# B&R Automation Studio project NAEUL004C00R13L518F00 (part 41)

#### Act_InputConfig.st
```iecst
(** 2019-04-09 **)
ACTION Act_InputConfig:

	(* Always Change If Project Change *)

	//Pass Data To Link
	tylocalPneu.In.bLinkDIConvClrSen := g_tyDInput.bConvClrSen;
	tylocalPneu.In.bConvPusherReachedRetSlw := g_tyPshrConv.bPshrRetAllwTrav;
	tylocalPneu.In.bLinkDIPusherRetRS := g_tyDInput.bPusherRetRS;
	tylocalPneu.In.eLinkLifterBtmStat := g_tyLifterBtm.eStat;
	tylocalPneu.In.eLinkLifterBtmStatus := g_tyLifterBtm.eStatus;
	tylocalPneu.In.eLinkLifter2Stat := g_tyLifter2.eStat;
	tylocalPneu.In.eLinkLifter2Status := g_tyLifter2.eStatus;

	//Pass Data To Internal Use
	tylocalPneu.In.bSafetyRelaySig 	 	 := g_tyDInput.bSafetyRlySig;
	tylocalPneu.In.udiRstErr := g_tyRstErr.udiReset;
	tylocalPneu.In.bPrep := g_tyNtParamCurr.bProjOutletShutPrep;
	tylocalPneu.In.bUISimu := g_tyUIOut.bSimuMod;
	tylocalPneu.In.bManual := g_tyUIOut.bMnlMod;
	tylocalPneu.In.bTwoCtrlIn := g_tyNtParamCurr.bOutShutterTwoCtrlIn;
	tylocalPneu.In.sProgNm := g_tyNtParamCurr.sOutShutterProgNm;
	tylocalPneu.In.bExtSen := g_tyDInput.bOutShutterCloseRS;
	tylocalPneu.In.bRetSen := g_tyDInput.bOutShutterOpenRS;
	tylocalPneu.In.tExtTO := g_tyNtParamCurr.tOutShutterExtTO;
	tylocalPneu.In.tRetTO := g_tyNtParamCurr.tOutShutterRetTO;
	tylocalPneu.In.bNtParamProjLifter2Prep := g_tyNtParamProjLifter2Prep;
	tylocalPneu.In.ePneuSel				 := Pneu2Sen; //Pneumatic With 2 Sensors
	(* Always Change If Project Change *)

	tylocalPneu.In.bExtSafetySen := (tylocalPneu.In.bLinkDIConvClrSen = FALSE) AND (tylocalPneu.In.bLinkDIPusherRetRS OR tylocalPneu.In.bConvPusherReachedRetSlw);

	IF g_tyOps.bRun = TRUE THEN
		IF tylocalPneu.In.bNtParamProjLifter2Prep = FALSE  THEN
			IF tylocalPneu.In.eLinkLifterBtmStat = LifterActIdle AND tylocalPneu.In.eLinkLifterBtmStatus <> Busy  THEN //
				tylocalPneu.In.eAct := g_tyOpsTravLifUL.eOutletPneuAct;
			ELSE
				tylocalPneu.In.eAct := eAct;
			END_IF
		ELSE
			IF tylocalPneu.In.eLinkLifterBtmStat = LifterActIdle AND tylocalPneu.In.eLinkLifterBtmStatus <> Busy AND tylocalPneu.In.eLinkLifter2Stat = LifterActIdle AND tylocalPneu.In.eLinkLifter2Status <> Busy  THEN // tylocalPneu.In.eLinkLifter2Status <> Busy
				tylocalPneu.In.eAct := g_tyOpsTravLifUL.eOutletPneuAct;
			ELSE
				tylocalPneu.In.eAct := eAct;
			END_IF
		END_IF
	ELSIF tylocalPneu.In.bManual = TRUE OR tylocalPneu.In.bUISimu THEN
		tylocalPneu.In.eAct := g_tyUIOut.eMnlAct.eOutShutterAct;
	ELSIF tylocalPneu.In.bSimu THEN
		tylocalPneu.In.eAct := g_tySimu1.eOutShutterAct;
	ELSE
		tylocalPneu.In.eAct := eAct;
	END_IF

END_ACTION
```

#### Act_OutputConfig.st
```iecst
ACTION Act_OutputConfig:

	// Output: Assign To Global For Independent Package Usage

	g_tyPneuOutShutter := tylocalPneu.Out; // Change the Global Naming According to the Physical Hardware Module

END_ACTION
```

### Program Logical/Pneu/PneuOutShutter2 (IEC, version 1.00.0) - 1.00.0 - NtPneu v5.00.0

#### Act_InputConfig.st - Change By Project
```iecst
(** 2019-04-09 **)
ACTION Act_InputConfig:

	(* Always Change If Project Change *)

	//Pass Data To Link
	tylocalPneu.In.bLinkDIConvClrSen := g_tyDInput.bConvClrSen;
	tylocalPneu.In.bConvPusherReachedRetSlw := g_tyPshrConv.bPshrRetAllwTrav;
	tylocalPneu.In.bLinkDIPusherRetRS := g_tyDInput.bPusherRetRS;
	tylocalPneu.In.eLinkLifterBtmStat := g_tyLifterBtm.eStat;
	tylocalPneu.In.eLinkLifterBtmStatus := g_tyLifterBtm.eStatus;
	tylocalPneu.In.eLinkLifter2Stat := g_tyLifter2.eStat;
	tylocalPneu.In.eLinkLifter2Status := g_tyLifter2.eStatus;

	//Pass Data To Internal Use
	tylocalPneu.In.bSafetyRelaySig 	 	 := g_tyDInput.bSafetyRlySig;
	tylocalPneu.In.udiRstErr := g_tyRstErr.udiReset;
	tylocalPneu.In.bPrep := g_tyNtParamCurr.bProjOutletShut2Prep;
	tylocalPneu.In.bUISimu := g_tyUIOut.bSimuMod;
	tylocalPneu.In.bManual := g_tyUIOut.bMnlMod;
	tylocalPneu.In.bTwoCtrlIn := g_tyNtParamCurr.bOutShutterTwoCtrlIn;
	tylocalPneu.In.sProgNm := g_tyNtParamCurr.sOutShutterProgNm;
	tylocalPneu.In.bExtSen := g_tyDInput.bOutShutterCloseRS2;
	tylocalPneu.In.bRetSen := g_tyDInput.bOutShutterOpenRS2;
	tylocalPneu.In.tExtTO := g_tyNtParamCurr.tOutShutterExtTO;
	tylocalPneu.In.tRetTO := g_tyNtParamCurr.tOutShutterRetTO;
	tylocalPneu.In.bNtParamProjLifter2Prep := g_tyNtParamProjLifter2Prep;
	tylocalPneu.In.ePneuSel				 := Pneu2Sen; //Pneumatic With 2 Sensors
	(* Always Change If Project Change *)
	tylocalPneu.In.bEn :=  g_tyNtParamCurr.bCurtainSenPrep;

	tylocalPneu.In.bExtSafetySen := (tylocalPneu.In.bLinkDIConvClrSen = FALSE) AND (tylocalPneu.In.bLinkDIPusherRetRS OR tylocalPneu.In.bConvPusherReachedRetSlw);

	IF g_tyOps.bRun = TRUE THEN
		IF tylocalPneu.In.bNtParamProjLifter2Prep = FALSE  THEN
			IF tylocalPneu.In.eLinkLifterBtmStat = LifterActIdle AND tylocalPneu.In.eLinkLifterBtmStatus <> Busy  THEN //
				tylocalPneu.In.eAct := g_tyOpsTravLifUL.eOutletPneuAct2;
			ELSE
				tylocalPneu.In.eAct := eAct;
			END_IF
		ELSE
			IF tylocalPneu.In.eLinkLifterBtmStat = LifterActIdle AND tylocalPneu.In.eLinkLifterBtmStatus <> Busy AND tylocalPneu.In.eLinkLifter2Stat = LifterActIdle AND tylocalPneu.In.eLinkLifter2Status <> Busy  THEN // tylocalPneu.In.eLinkLifter2Status <> Busy
				tylocalPneu.In.eAct := g_tyOpsTravLifUL.eOutletPneuAct2;
			ELSE
				tylocalPneu.In.eAct := eAct;
			END_IF
		END_IF
	ELSIF tylocalPneu.In.bManual = TRUE OR tylocalPneu.In.bUISimu THEN
		tylocalPneu.In.eAct := g_tyUIOut.eMnlAct.eOutShutterAct2;
	ELSIF tylocalPneu.In.bSimu THEN
		tylocalPneu.In.eAct := g_tySimu1.eOutShutterAct2;
	ELSE
		tylocalPneu.In.eAct := eAct;
	END_IF
END_ACTION
```

#### Act_OutputConfig.st - Change By Project
```iecst
ACTION Act_OutputConfig:

	(* Always Change If Project Change *)

	//Pass Address To Global Address For External Use
	//Action, State & Status
	p_Pneu2SenOutShutterStat2		:= ADR(eStat);
	p_Pneu2SenOutShutterStatus2		:= ADR(eStatus);
	p_Pneu2SenOutShutterStatTxt2	:= ADR(sStatTxt);

	//Alarm
	p_Pneu2SenOutShutterAlmData2	:= ADR(tyAlmData);

	//Output
	p_Pneu2SenOutShutterExtCtrl2	:= ADR(bExtCtrl);
	p_Pneu2SenOutShutterRetCtrl2	:= ADR(bRetCtrl);
	p_Pneu2SenOutShutterTwoCtrlOut2	:= ADR(bTwoCtrlOut);
	p_Pneu2SenOutShutterExtended2	:= ADR(bExtended);
	p_Pneu2SenOutShutterRetracted2	:= ADR(bRetracted);

END_ACTION
```

### Program Logical/Pneu/PneuOutShutter3 (IEC) - 1.00.0 - NtPneu v5.00.0

#### Act_Alarm.st
```iecst
ACTION Act_Alarm:

	// Reset Error
	IF tylocalPneu.In.udiRstErr <> udiRstErrOld THEN
		bRstErr			:= TRUE;
		udiRstErrOld	:= tylocalPneu.In.udiRstErr;
	ELSE
		bRstErr			:= FALSE;
	END_IF

	//Error State
	IF (tylocalPneu.Out.eStatus = Error) AND bRstErr THEN
		tylocalPneu.In.eAct		:= PneuActIdle; //Command Action From Global
		tylocalPneu.Out.eStat	:= PneuActIdle; //Feedback State To Global
	END_IF

	//Error Link To HMI
	IF EDGEPOS(tylocalPneu.Out.eStatus = Error) THEN

		tylocalPneu.Out.tyAlmData.udiCode		:= udiStatus;
		tylocalPneu.Out.tyAlmData.eSeverity		:= AlmSeverityError;
		tylocalPneu.Out.tyAlmData.udiRunTime	:= tylocalPneu.Out.tyAlmData.udiRunTime + 1;
		tylocalPneu.Out.tyAlmData.bAlm			:= TRUE;
		tylocalPneu.Out.tyAlmData.udiModuleNum  := udiModuleNum;
		g_tyAlmProgNm.sPneuShutterProgNm		:= tylocalPneu.In.sProgNm;

	ELSIF bRstErr AND (tylocalPneu.Out.tyAlmData.udiCode <> 0) THEN

		tylocalPneu.Out.tyAlmData.udiCode	:= 0;
		tylocalPneu.Out.tyAlmData.eSeverity	:= AlmSeverityNA;
		tylocalPneu.Out.tyAlmData.bAlm		:= FALSE;

	END_IF

END_ACTION
```

#### Act_OutputConfig.st
```iecst
(** 2019-03-25 **)
PROGRAM _INIT

	(* Always Change If Project Change *)

	//Pass Address To Global Address For External Use
	//Action, State & Status
	p_Pneu2SenOutShutterStat3			:= ADR(eStat);
	p_Pneu2SenOutShutterStatus3			:= ADR(eStatus);
	p_Pneu2SenOutShutterStatTxt3		:= ADR(sStatTxt);

	//Alarm
	p_Pneu2SenOutShutterAlmData3		:= ADR(tyAlmData);

	//Output
	p_Pneu2SenOutShutterExtCtrl3		:= ADR(bExtCtrl);
	p_Pneu2SenOutShutterRetCtrl3		:= ADR(bRetCtrl);
	p_Pneu2SenOutShutterTwoCtrlOut3		:= ADR(bTwoCtrlOut);
	p_Pneu2SenOutShutterExtended3		:= ADR(bExtended);
	p_Pneu2SenOutShutterRetracted3		:= ADR(bRetracted);

	(* Always Change If Project Change *)

END_PROGRAM
```

### Program Logical/Pneu/PneuStopperA (IEC) - 1.00.0 - NtPneu v5.00.0

#### Act_InputConfig.st
```iecst
(** 2019-04-09 **)
ACTION Act_InputConfig:

	(* Always Change If Project Change *)

	//Pass Data To Link

	tylocalPneu.In.bSafetyRelaySig 	 	 := g_tyDInput.bSafetyRlySig;
	tylocalPneu.In.udiRstErr		 	 := g_tyRstErrOut.udiRstErr;
	tylocalPneu.In.bPrep			  	 := g_tyNtParamCurr.bProjStopperAPrep;
	tylocalPneu.In.bDis			  	 	 := g_tyMcParamCurr.bStopperADis;

	tylocalPneu.In.bManual		  	 	 := g_tyUIOut.bUIManualMod;
	tylocalPneu.In.bTwoCtrlIn		 	 := g_tyNtParamCurr.bStopperATwoCtrlIn;
	tylocalPneu.In.sProgNm			 	 := g_tyNtParamCurr.sStopperAProgNm;

	tylocalPneu.In.tExtTO			 	 := g_tyNtParamCurr.tStopperAExtDlyTm;
	tylocalPneu.In.tRetTO		 	     := g_tyNtParamCurr.tStopperARetDlyTm ;
	tylocalPneu.In.ePneuSel				 := PneuNoSen; //Pneumatic With 2 Sensors

	IF g_tyOps.bRun = TRUE THEN
		tylocalPneu.In.eAct := g_tyOpsTravLifUL.eStopperAct1;
	ELSIF tylocalPneu.In.bManual = TRUE OR tylocalPneu.In.bUISimu THEN
		tylocalPneu.In.eAct := g_tyUIOut.eMnlAct.eStopperAAct;
	ELSE
		tylocalPneu.In.eAct := eAct;
	END_IF

END_ACTION
```

#### Act_OutputConfig.st
```iecst
(** 2019-03-25 **)
ACTION Act_OutputConfig:
		// Output: Assign To Global For Independent Package Usage

	g_tyPneuStopperA := tylocalPneu.Out; // Change the Global Naming According to the Physical Hardware Module

END_ACTION
```

### Program Logical/Pneu/PneuStopperB (IEC) - 1.00.0 - NtPneu v5.00.0

#### Act_InputConfig.st
```iecst
(** 2019-04-09 **)
ACTION Act_InputConfig:

	(* Always Change If Project Change *)

	//Pass Data To Link

	tylocalPneu.In.bSafetyRelaySig 	 	 := g_tyDInput.bSafetyRlySig;
	tylocalPneu.In.udiRstErr		 	 := g_tyRstErrOut.udiRstErr;
	tylocalPneu.In.bPrep			  	 := g_tyNtParamCurr.bProjStopperBPrep;
	tylocalPneu.In.bDis			  	 	 := g_tyMcParamCurr.bStopperBDis;

	tylocalPneu.In.bManual		  	 	 := g_tyUIOut.bUIManualMod;
	tylocalPneu.In.bTwoCtrlIn		 	 := g_tyNtParamCurr.bStopperBTwoCtrlIn;
	tylocalPneu.In.sProgNm			 	 := g_tyNtParamCurr.sStopperBProgNm;

	tylocalPneu.In.tExtTO			 	 := g_tyNtParamCurr.tStopperBExtDlyTm;
	tylocalPneu.In.tRetTO		 	     := g_tyNtParamCurr.tStopperBRetDlyTm ;
	tylocalPneu.In.ePneuSel				 := PneuNoSen; //Pneumatic With 2 Sensors

	IF g_tyOps.bRun = TRUE THEN
		tylocalPneu.In.eAct := g_tyOpsTravLifUL.eStopperAct2;
	ELSIF tylocalPneu.In.bManual = TRUE OR tylocalPneu.In.bUISimu THEN
		tylocalPneu.In.eAct := g_tyUIOut.eMnlAct.eStopperBAct;
	ELSE
		tylocalPneu.In.eAct := eAct;
	END_IF

END_ACTION
```

#### Act_OutputConfig.st
```iecst
(** 2019-03-25 **)
ACTION Act_OutputConfig:
		// Output: Assign To Global For Independent Package Usage

	g_tyPneuStopperB := tylocalPneu.Out; // Change the Global Naming According to the Physical Hardware Module

END_ACTION
```

### Program Logical/Pneu/PneuStopperC (IEC) - 1.00.0 - NtPneu v5.00.0

#### Act_InputConfig.st
```iecst
(** 2019-04-09 **)
ACTION Act_InputConfig:

	(* Always Change If Project Change *)

	//Pass Data To Link

	tylocalPneu.In.bSafetyRelaySig 	 	 := g_tyDInput.bSafetyRlySig;
	tylocalPneu.In.udiRstErr		 	 := g_tyRstErrOut.udiRstErr;
	tylocalPneu.In.bPrep			  	 := g_tyNtParamCurr.bProjStopperCPrep;
	tylocalPneu.In.bDis			  	 	 := g_tyMcParamCurr.bStopperCDis;

	tylocalPneu.In.bManual		  	 	 := g_tyUIOut.bUIManualMod;
	tylocalPneu.In.bTwoCtrlIn		 	 := g_tyNtParamCurr.bStopperCTwoCtrlIn;
	tylocalPneu.In.sProgNm			 	 := g_tyNtParamCurr.sStopperCProgNm;

	tylocalPneu.In.tExtTO			 	 := g_tyNtParamCurr.tStopperCExtDlyTm;
	tylocalPneu.In.tRetTO		 	     := g_tyNtParamCurr.tStopperCRetDlyTm ;
	tylocalPneu.In.ePneuSel				 := PneuNoSen; //Pneumatic With 2 Sensors

	IF g_tyOps.bRun = TRUE THEN
		tylocalPneu.In.eAct := g_tyOpsTravLifUL.eStopperAct3;
	ELSIF tylocalPneu.In.bManual = TRUE OR tylocalPneu.In.bUISimu THEN
		tylocalPneu.In.eAct := g_tyUIOut.eMnlAct.eStopperCAct;
	ELSE
		tylocalPneu.In.eAct := eAct;
	END_IF

END_ACTION
```

#### Act_Main.st
```iecst
ACTION Act_Main:

	IF tylocalPneu.In.bSafetyRelaySig = FALSE OR EDGEPOS(tylocalPneu.Out.eStatus = Error) THEN
		tylocalPneu.Out.bExtCtrl 	:= FALSE;
		tylocalPneu.Out.bRetCtrl 	:= FALSE;
		tylocalPneu.Out.bExtended	:= FALSE;
		tylocalPneu.Out.bRetracted  := FALSE;
	END_IF

	//Execution Action
	IF tylocalPneu.Out.eStatus <> Error THEN
		tylocalPneu.Out.eStat := tylocalPneu.In.eAct;
	END_IF

	//Transition State
	IF eStatOld <> tylocalPneu.Out.eStat THEN

		fbPneuNoSenExt(bEn := FALSE);
		fbPneuNoSenRet(bEn := FALSE);

		fbPneu2SenExt(bEn := FALSE);
		fbPneu2SenRet(bEn := FALSE);

		eStatOld	:= tylocalPneu.Out.eStat;

		tylocalPneu.Out.eStatus		:= Busy;
	END_IF

	//Main
	CASE tylocalPneu.Out.eStat OF

		PneuActIdle:
			tylocalPneu.Out.eStatus	:= Idle;

		PneuActSetAll:
			IF tylocalPneu.Out.eStatus = Idle OR tylocalPneu.Out.eStatus = Busy THEN

				fbPneuNoSenExt(bEn := FALSE);
				fbPneuNoSenRet(bEn := FALSE);

				fbPneu2SenExt(bEn := FALSE);
				fbPneu2SenRet(bEn := FALSE);

				tylocalPneu.Out.bExtCtrl	:= TRUE;
				tylocalPneu.Out.bRetCtrl	:= TRUE;

				tylocalPneu.Out.bExtended	:= FALSE;
				tylocalPneu.Out.bRetracted	:= FALSE;

				tylocalPneu.Out.eStatus	:= Done;

			END_IF

		PneuActRstAll:
			IF tylocalPneu.Out.eStatus = Idle OR tylocalPneu.Out.eStatus = Busy THEN

				fbPneuNoSenExt(bEn := FALSE);
				fbPneuNoSenRet(bEn := FALSE);

				fbPneu2SenExt(bEn := FALSE);
				fbPneu2SenRet(bEn := FALSE);

				tylocalPneu.Out.bExtCtrl	:= FALSE;
				tylocalPneu.Out.bRetCtrl	:= FALSE;

				tylocalPneu.Out.bExtended	:= FALSE;
				tylocalPneu.Out.bRetracted	:= FALSE;

				tylocalPneu.Out.eStatus	:= Done;

			END_IF

		PneuActSetExt:
			IF tylocalPneu.Out.eStatus = Idle OR tylocalPneu.Out.eStatus = Busy THEN

				fbPneuNoSenExt(bEn := FALSE);
				fbPneuNoSenRet(bEn := FALSE);

				fbPneu2SenExt(bEn := FALSE);
				fbPneu2SenRet(bEn := FALSE);

				tylocalPneu.Out.bExtCtrl	:= TRUE;
				tylocalPneu.Out.bRetCtrl	:= FALSE;

				tylocalPneu.Out.bExtended	:= TRUE;
				tylocalPneu.Out.bRetracted	:= FALSE;

				tylocalPneu.Out.eStatus	:= Done;

			END_IF

		PneuActSetRet:
			IF tylocalPneu.Out.eStatus = Idle OR tylocalPneu.Out.eStatus = Busy THEN

				//Reset
				fbPneuNoSenExt(bEn := FALSE);
				fbPneuNoSenRet(bEn := FALSE);

				fbPneu2SenExt(bEn := FALSE);
				fbPneu2SenRet(bEn := FALSE);

				tylocalPneu.Out.bExtCtrl	:= FALSE;
				tylocalPneu.Out.bRetCtrl	:= TRUE;

				tylocalPneu.Out.bExtended	:= FALSE;
				tylocalPneu.Out.bRetracted	:= TRUE;

				tylocalPneu.Out.eStatus	:= Done;

			END_IF

		PneuActExt:
			IF tylocalPneu.Out.eStatus = Idle OR tylocalPneu.Out.eStatus = Busy THEN

				tylocalPneu.Out.eStatus	:= Busy;

				tylocalPneu.Out.bExtCtrl	:= TRUE;
				tylocalPneu.Out.bRetCtrl	:= FALSE;

				CASE tylocalPneu.In.ePneuSel OF

					PneuNoSen: //Pneumatic Without Sen // 0
						fbPneuNoSenExt.bExtSafety	:= tylocalPneu.In.bExtSafetySen;
						fbPneuNoSenExt.tDlyTm		:= tylocalPneu.In.tExtDlyTm;
						fbPneuNoSenExt(bEn := TRUE);
					Pneu2Sen: //Pneumatic With 2 Sen // 3
						fbPneu2SenExt.bExtSen   	:= tylocalPneu.In.bExtSen;
						fbPneu2SenExt.bRetSen   	:= tylocalPneu.In.bRetSen;
						fbPneu2SenExt.bExtSafety	:= tylocalPneu.In.bExtSafetySen;
						fbPneu2SenExt.tTimeOut		:= tylocalPneu.In.tExtTO;
						fbPneu2SenExt(bEn := TRUE);
				END_CASE

				IF fbPneuNoSenExt.udiStatus = 0 OR
					fbPneu2SenExt.udiStatus = 0 THEN

					tylocalPneu.Out.bExtended	:= TRUE;
					tylocalPneu.Out.bRetracted	:= FALSE;
					tylocalPneu.Out.eStatus		:= Done;

				ELSIF (fbPneuNoSenExt.udiStatus > 0 AND fbPneuNoSenExt.udiStatus < 65534) OR
					(fbPneu2SenExt.udiStatus > 0 AND fbPneu2SenExt.udiStatus < 65534) THEN

					IF tylocalPneu.In.bTwoCtrlIn = TRUE THEN

						tylocalPneu.Out.bExtCtrl	:= FALSE;
						tylocalPneu.Out.bRetCtrl	:= FALSE;

					ELSE
						tylocalPneu.Out.bExtCtrl	:= FALSE;
						tylocalPneu.Out.bRetCtrl	:= TRUE;

					END_IF

					tylocalPneu.Out.bExtended	:= FALSE;
					tylocalPneu.Out.bRetracted	:= FALSE;

					tylocalPneu.Out.eStatus		:= Error;

					IF fbPneuNoSenExt.udiStatus = 1507 OR fbPneu2SenExt.udiStatus  = 1507 THEN
						udiStatus	:= 2401; //Safety Check Error While Extending
					ELSIF fbPneu2SenExt.udiStatus = 1503 THEN
						udiStatus	:= 2552;	//Extend Sensor On Checking Time Out While Extending
					ELSIF fbPneu2SenExt.udiStatus = 1506 THEN
						udiStatus	:= 2553; //Retract Sensor Off Checking Time Out While Extending
					ELSE
						IF tylocalPneu.In.ePneuSel = PneuNoSen THEN
							udiStatus	:= fbPneuNoSenExt.udiStatus;
						ELSE
							udiStatus	:= fbPneu2SenExt.udiStatus;
						END_IF
					END_IF
				END_IF

			END_IF

		PneuActRet:
			IF tylocalPneu.Out.eStatus = Idle OR tylocalPneu.Out.eStatus = Busy THEN

				tylocalPneu.Out.eStatus	:= Busy;

				tylocalPneu.Out.bExtCtrl	:= FALSE;
				tylocalPneu.Out.bRetCtrl	:= TRUE;

				CASE tylocalPneu.In.ePneuSel OF

					PneuNoSen: //Pneumatic Without Sen // 0
						fbPneuNoSenRet.bRetSafety	:= tylocalPneu.In.bRetSafetySen;
						fbPneuNoSenRet.tDlyTm		:= tylocalPneu.In.tRetDlyTm;
						fbPneuNoSenRet(bEn := TRUE);
					Pneu2Sen: //Pneumatic With 2 Sen // 3
						fbPneu2SenRet.bExtSen   	:= tylocalPneu.In.bExtSen;
						fbPneu2SenRet.bRetSen   	:= tylocalPneu.In.bRetSen;
						fbPneu2SenRet.bRetSafety	:= tylocalPneu.In.bRetSafetySen;
						fbPneu2SenRet.tTimeOut		:= tylocalPneu.In.tRetTO;
						fbPneu2SenRet(bEn := TRUE);
				END_CASE

				IF fbPneuNoSenRet.udiStatus = 0 OR
					fbPneu2SenRet.udiStatus = 0 THEN

					tylocalPneu.Out.bExtended	:= FALSE;
					tylocalPneu.Out.bRetracted	:= TRUE;
					tylocalPneu.Out.eStatus		:= Done;

				ELSIF (fbPneuNoSenRet.udiStatus > 0 AND fbPneuNoSenRet.udiStatus < 65534) OR
					(fbPneu2SenRet.udiStatus > 0 AND fbPneu2SenRet.udiStatus < 65534) THEN

					IF tylocalPneu.In.bTwoCtrlIn = TRUE THEN
						tylocalPneu.Out.bExtCtrl	:= FALSE;
						tylocalPneu.Out.bRetCtrl	:= FALSE;
					ELSE
						tylocalPneu.Out.bExtCtrl	:= TRUE;
						tylocalPneu.Out.bRetCtrl	:= FALSE;
					END_IF

					tylocalPneu.Out.bExtended	:= FALSE;
					tylocalPneu.Out.bRetracted	:= FALSE;

					tylocalPneu.Out.eStatus		:= Error;

					IF fbPneuNoSenRet.udiStatus = 1508 OR fbPneu2SenRet.udiStatus = 1508 THEN
						udiStatus	:= 2404;	//Safety Check Error While Retracting
					ELSIF fbPneu2SenRet.udiStatus = 1505 THEN
						udiStatus	:= 2555;	//Retract Sensor On Checking Time Out While Retracting
					ELSIF fbPneu2SenRet.udiStatus = 1504 THEN
						udiStatus	:= 2556;    //Extend Sensor Off Checking Time Out While Retracting
					ELSE
						IF tylocalPneu.In.ePneuSel = PneuNoSen THEN
							udiStatus	:= fbPneuNoSenRet.udiStatus;
						ELSE
							udiStatus	:= fbPneu2SenRet.udiStatus;
						END_IF
					END_IF
				END_IF

			END_IF

		ELSE
			IF tylocalPneu.Out.eStatus = Idle OR tylocalPneu.Out.eStatus = Busy THEN
				tylocalPneu.Out.eStatus	:= Done;
			END_IF

	END_CASE

	//background
	IF tylocalPneu.In.ePneuSel = Pneu2Sen THEN
		IF tylocalPneu.In.bExtSen = FALSE THEN
			tylocalPneu.Out.bExtended	:= FALSE;
		END_IF

		IF tylocalPneu.In.bRetSen = FALSE THEN
			tylocalPneu.Out.bRetracted	:= FALSE;
		END_IF
	END_IF

END_ACTION
```

#### Act_OutputConfig.st
```iecst
(** 2019-03-25 **)
ACTION Act_OutputConfig:
		// Output: Assign To Global For Independent Package Usage

		g_tyPneuStopperC := tylocalPneu.Out; // Change the Global Naming According to the Physical Hardware Module

END_ACTION
```

### Program Logical/Pneu/PneuSelClamp1 (IEC) - 1.00.0 - NtPneu v5.00.0

#### Act_InputConfig.st
```iecst
(** 2019-04-09 **)
ACTION Act_InitGlobal:

	(* Always Change If Project Change *)

	//Pass Data To Link
	p_bLinkDISafetyRlySig				 := g_tyDISafetyRlySig;
	tylocalPneu.In.udiRstErr		 	 := g_tyRstErrOut.udiRstErr;
	tylocalPneu.In.bPrep 	 			 := g_tyNtParamCurr.bMagAutoVerifyPrep;
	tylocalPneu.In.bManual		  	 	 := g_tyUIOut.bUIManualMod;
	tylocalPneu.In.bTwoCtrlIn		 	 := g_tyNtParamCurr.bSelClamp1TwoCtrlIn;
	tylocalPneu.In.sProgNm			 	 := g_tyNtParamCurr.sSelClamp1ProgNm;
	tylocalPneu.In.bExtSen 				 := g_tyDIMag1SelUnclampRS;
	//tylocalPneu.In.bRetSen := g_tyDIOutShutterOpenRS;
	tylocalPneu.In.tExtTO 				 := g_tyNtParamCurr.SelClamp1ExtDlyTm;
	tylocalPneu.In.tRetTO 				 := g_tyNtParamCurr.SelClamp1RetDlyTm;
	tylocalPneu.In.ePneuSel				 := Pneu2Sen;
	(* Always Change If Project Change *)
	tylocalPneu.In.bRetSen := NOT(tylocalPneu.In.bExtSen);

	IF g_tyOps.bRun = TRUE THEN
		tylocalPneu.In.eAct := g_tyOpsMagConvUL1.eSelClampCtrl;
	ELSIF tylocalPneu.In.bManual = TRUE THEN
		tylocalPneu.In.eAct := g_tyUIOut.eMnlAct.eMagConvSelClp1Act;
	ELSE
		tylocalPneu.In.eAct := eAct;
	END_IF
END_ACTION
```

#### Act_OutputConfig.st
```iecst
ACTION Act_OutputConfig:
	// Output: Assign To Global For Independent Package Usage

	g_tyPneuSelClamp1 := tylocalPneu.Out; // Change the Global Naming According to the Physical Hardware Module

END_ACTION
```

### Program Logical/Pneu/PneuSelClamp2 (IEC) - 1.00.0 - NtPneu v5.00.0

#### Act_InputConfig.st
```iecst
(** 2019-04-09 **)
ACTION Act_InitGlobal:

	(* Always Change If Project Change *)

	//Pass Data To Link
	p_bLinkDISafetyRlySig				 := g_tyDISafetyRlySig;
	tylocalPneu.In.udiRstErr		 	 := g_tyRstErrOut.udiRstErr;
	tylocalPneu.In.bPrep 	 			 := g_tyNtParamCurr.bMagAutoVerifyPrep;
	tylocalPneu.In.bManual		  	 	 := g_tyUIOut.bUIManualMod;
	tylocalPneu.In.bTwoCtrlIn		 	 := g_tyNtParamCurr.bSelClamp2TwoCtrlIn;
	tylocalPneu.In.sProgNm			 	 := g_tyNtParamCurr.sSelClamp2ProgNm;
	tylocalPneu.In.bExtSen			 	 := g_tyDIMag2SelUnclampRS;
	//tylocalPneu.In.bRetSen := g_tyDIOutShutterOpenRS;
	tylocalPneu.In.tExtTO 				 := g_tyNtParamCurr.SelClamp2ExtDlyTm;
	tylocalPneu.In.tRetTO 				 := g_tyNtParamCurr.SelClamp2RetDlyTm;
	tylocalPneu.In.ePneuSel				 := Pneu2Sen;
	(* Always Change If Project Change *)
	tylocalPneu.In.bRetSen := NOT(tylocalPneu.In.bExtSen);

	IF g_tyOps.bRun = TRUE THEN
		tylocalPneu.In.eAct := g_tyOpsMagConvUL2.eSelClampCtrl;
	ELSIF tylocalPneu.In.bManual = TRUE THEN
		tylocalPneu.In.eAct := g_tyUIOut.eMnlAct.eMagConvSelClp2Act;
	ELSE
		tylocalPneu.In.eAct := eAct;
	END_IF
END_ACTION
```

#### Act_OutputConfig.st
```iecst
ACTION Act_OutputConfig:
	// Output: Assign To Global For Independent Package Usage

	g_tyPneuSelClamp2 := tylocalPneu.Out; // Change the Global Naming According to the Physical Hardware Module

END_ACTION
```

### Program Logical/Pneu/PneuSelClamp3 (IEC) - 1.00.0 - NtPneu v5.00.0

#### Act_InputConfig.st
```iecst
(** 2019-04-09 **)
ACTION Act_InitGlobal:

	(* Always Change If Project Change *)

	//Pass Data To Link
	p_bLinkDISafetyRlySig 				 := g_tyDISafetyRlySig;
	tylocalPneu.In.udiRstErr		 	 := g_tyRstErrOut.udiRstErr;
	tylocalPneu.In.bPrep 	 			 := g_tyNtParamCurr.bMagAutoVerifyPrep;
	tylocalPneu.In.bManual		  	 	 := g_tyUIOut.bUIManualMod;
	tylocalPneu.In.bTwoCtrlIn		 	 := g_tyNtParamCurr.bSelClamp3TwoCtrlIn;
	tylocalPneu.In.sProgNm			 	 := g_tyNtParamCurr.sSelClamp3ProgNm;
	tylocalPneu.In.bExtSen 				 := g_tyDIMag3SelUnclampRS;
	//tylocalPneu.In.bRetSen := g_tyDIOutShutterOpenRS;
	tylocalPneu.In.tExtTO 				 := g_tyNtParamCurr.SelClamp3ExtDlyTm;
	tylocalPneu.In.tRetTO 				 := g_tyNtParamCurr.SelClamp3RetDlyTm;
	tylocalPneu.In.ePneuSel				 := Pneu2Sen;
	(* Always Change If Project Change *)
	tylocalPneu.In.bRetSen := NOT(tylocalPneu.In.bExtSen);

	IF g_tyOps.bRun = TRUE THEN
		tylocalPneu.In.eAct := g_tyOpsMagConvUL3.eSelClampCtrl;
	ELSIF tylocalPneu.In.bManual = TRUE THEN
		tylocalPneu.In.eAct := g_tyUIOut.eMnlAct.eMagConvSelClp3Act;
	ELSE
		tylocalPneu.In.eAct := eAct;
	END_IF
END_ACTION
```

#### Act_OutputConfig.st
```iecst
ACTION Act_OutputConfig:
	// Output: Assign To Global For Independent Package Usage

	g_tyPneuSelClamp3 := tylocalPneu.Out; // Change the Global Naming According to the Physical Hardware Module

END_ACTION
```

### Program Logical/Pneu/PneuMag1SafetyBar (IEC) - 1.00.0 - NtPneu v5.00.0

#### Act_InputConfig.st
```iecst
ACTION Act_InputConfig:

	(* Always Change If Project Change *)

	tylocalPneu.In.bSafetyRelaySig 	 	 := g_tyDInput.bSafetyRlySig;
	tylocalPneu.In.bMagRcpCurrRcpSBarDisabled ACCESS p_MagRcpCurrRcpSBarDisabled;

	//Pass Data To Internal Use
	tylocalPneu.In.udiRstErr		 	 := g_tyRstErrOut.udiRstErr;
	tylocalPneu.In.bPrep := g_tyNtParamCurr.bProjMagSafetyBarPrep;
//	tylocalPneu.In.bDis := g_tyMcParamMagAWDis;
	tylocalPneu.In.bManual := g_tyUIOut.bUIManualMod;
	tylocalPneu.In.bTwoCtrlIn := g_tyNtParamCurr.bMag1SafetyBarTwoCtrlIn;
	tylocalPneu.In.sProgNm := g_tyNtParamCurr.sMag1SafetyBarProgNm;
	tylocalPneu.In.bExtSen := g_tyDIMag1SafetyBarExtRS;
	tylocalPneu.In.bRetSen := g_tyDIMag1SafetyBarRetRS;
	tylocalPneu.In.tExtTO := g_tyNtParamCurr.tMag1SafetyBarExtTO;
	tylocalPneu.In.tRetTO := g_tyNtParamCurr.tMag1SafetyBarRetTO;
	tylocalPneu.In.bNtSettingsLoadDone := g_tyStartupNtSettingsLoadDone;
	tylocalPneu.In.ePneuSel				 := Pneu2Sen;

	//Link bPrep, bEn & bDis
	IF g_tyStartUp.bRun AND tylocalPneu.In.bPrep THEN
		tylocalPneu.In.bDis := tylocalPneu.In.bMagRcpCurrRcpSBarDisabled;
	ELSE
		tylocalPneu.In.bDis := FALSE;
	END_IF

	IF g_tyOps.bRun = TRUE THEN
		tylocalPneu.In.eAct := g_tyOpsMagConvUL1.eSafetyBarAct;
	ELSIF tylocalPneu.In.bManual = TRUE THEN
		tylocalPneu.In.eAct := g_tyUIOut.eMnlAct.eMag1SafetyBarAct;
	ELSE
		tylocalPneu.In.eAct := eAct;
	END_IF

END_ACTION
```

#### Act_OutputConfig.st
```iecst
ACTION Act_OutputConfig:
	// Output: Assign To Global For Independent Package Usage

	g_tyPneuMag1SafetyBar := tylocalPneu.Out; // Change the Global Naming According to the Physical Hardware Module

END_ACTION
```

### Program Logical/Pneu/PneuMag2SafetyBar (IEC) - 1.00.0 - NtPneu v5.00.0

#### Act_InputConfig.st
```iecst
ACTION Act_InputConfig:

	(* Always Change If Project Change *)

	tylocalPneu.In.bSafetyRelaySig 	 	 := g_tyDInput.bSafetyRlySig;
	tylocalPneu.In.bMagRcpCurrRcpSBarDisabled ACCESS p_MagRcpCurrRcpSBarDisabled;

	//Pass Data To Internal Use
	tylocalPneu.In.udiRstErr		 	 := g_tyRstErrOut.udiRstErr;
	tylocalPneu.In.bPrep := g_tyNtParamCurr.bProjMagSafetyBarPrep;
//	tylocalPneu.In.bDis := g_tyMcParamMagAWDis;
	tylocalPneu.In.bManual := g_tyUIOut.bUIManualMod;
	tylocalPneu.In.bTwoCtrlIn := g_tyNtParamCurr.bMag2SafetyBarTwoCtrlIn;
	tylocalPneu.In.sProgNm := g_tyNtParamCurr.sMag2SafetyBarProgNm;
	tylocalPneu.In.bExtSen := g_tyDIMag2SafetyBarExtRS;
	tylocalPneu.In.bRetSen := g_tyDIMag2SafetyBarRetRS;
	tylocalPneu.In.tExtTO := g_tyNtParamCurr.tMag2SafetyBarExtTO;
	tylocalPneu.In.tRetTO := g_tyNtParamCurr.tMag2SafetyBarRetTO;
	tylocalPneu.In.bNtSettingsLoadDone := g_tyStartupNtSettingsLoadDone;
	tylocalPneu.In.ePneuSel				 := Pneu2Sen;

	//Link bPrep, bEn & bDis
	IF g_tyStartUp.bRun AND tylocalPneu.In.bPrep THEN
		tylocalPneu.In.bDis := tylocalPneu.In.bMagRcpCurrRcpSBarDisabled;
	ELSE
		tylocalPneu.In.bDis := FALSE;
	END_IF

	IF g_tyOps.bRun = TRUE THEN
		tylocalPneu.In.eAct := g_tyOpsMagConvUL2.eSafetyBarAct;
	ELSIF tylocalPneu.In.bManual = TRUE THEN
		tylocalPneu.In.eAct := g_tyUIOut.eMnlAct.eMag2SafetyBarAct;
	ELSE
		tylocalPneu.In.eAct := eAct;
	END_IF

END_ACTION
```

#### Act_OutputConfig.st
```iecst
ACTION Act_OutputConfig:
	// Output: Assign To Global For Independent Package Usage

	g_tyPneuMag2SafetyBar := tylocalPneu.Out; // Change the Global Naming According to the Physical Hardware Module

END_ACTION
```

### Program Logical/Pneu/PneuMag3SafetyBar (IEC) - 1.00.0 - NtPneu v5.00.0

#### Act_InputConfig.st
```iecst
ACTION Act_InputConfig:

	(* Always Change If Project Change *)

	tylocalPneu.In.bSafetyRelaySig 	 	 := g_tyDInput.bSafetyRlySig;
	tylocalPneu.In.bMagRcpCurrRcpSBarDisabled ACCESS p_MagRcpCurrRcpSBarDisabled;

	//Pass Data To Internal Use
	tylocalPneu.In.udiRstErr		 	 := g_tyRstErrOut.udiRstErr;
	tylocalPneu.In.bPrep := g_tyNtParamCurr.bProjMagSafetyBarPrep;
//	tylocalPneu.In.bDis := g_tyMcParamMagAWDis;
	tylocalPneu.In.bManual := g_tyUIOut.bUIManualMod;
	tylocalPneu.In.bTwoCtrlIn := g_tyNtParamCurr.bMag3SafetyBarTwoCtrlIn;
	tylocalPneu.In.sProgNm := g_tyNtParamCurr.aMag3SafetyBarProgNm;
	tylocalPneu.In.bExtSen := g_tyDIMag3SafetyBarExtRS;
	tylocalPneu.In.bRetSen := g_tyDIMag3SafetyBarRetRS;
	tylocalPneu.In.tExtTO := g_tyNtParamCurr.tMag3SafetyBarExtTO;
	tylocalPneu.In.tRetTO := g_tyNtParamCurr.tMag3SafetyBarRetTO;
	tylocalPneu.In.bNtSettingsLoadDone := g_tyStartupNtSettingsLoadDone;
	tylocalPneu.In.ePneuSel				 := Pneu2Sen;

	//Link bPrep, bEn & bDis
	IF g_tyStartUp.bRun AND tylocalPneu.In.bPrep THEN
		tylocalPneu.In.bDis := tylocalPneu.In.bMagRcpCurrRcpSBarDisabled;
	ELSE
		tylocalPneu.In.bDis := FALSE;
	END_IF

	IF g_tyOps.bRun = TRUE THEN
		tylocalPneu.In.eAct := g_tyOpsMagConvUL3.eSafetyBarAct;
	ELSIF tylocalPneu.In.bManual = TRUE THEN
		tylocalPneu.In.eAct := g_tyUIOut.eMnlAct.eMag3SafetyBarAct;
	ELSE
		tylocalPneu.In.eAct := eAct;
	END_IF

END_ACTION
```

#### Act_OutputConfig.st
```iecst
ACTION Act_OutputConfig:
	// Output: Assign To Global For Independent Package Usage

	g_tyPneuMag1AWEngage:= tylocalPneu.Out; // Change the Global Naming According to the Physical Hardware Module

END_ACTION
```

### Program Logical/Pneu/PneuMag1AWEngage (IEC) - 1.00.0 - NtPneu v5.00.0

#### Act_InputConfig.st
```iecst
ACTION Act_InputConfig:

	(* Always Change If Project Change *)

	//Pass Data To Link
	tylocalPneu.In.bSafetyRelaySig 	 	 := g_tyDInput.bSafetyRlySig;
	tylocalPneu.In.udiRstErr		 	 := g_tyRstErrOut.udiRstErr;
	tylocalPneu.In.bPrep 				 := g_tyNtParamCurr.bProjMagAWPrep;
	tylocalPneu.In.bDis 				 := g_tyMcParamCurr.bMagAWDis;
	tylocalPneu.In.bManual 				 := g_tyUIOut.bUIManualMod;
	tylocalPneu.In.bTwoCtrlIn 			 := g_tyNtParamCurr.bMag1AWEngageTwoCtrlIn;
	tylocalPneu.In.sProgNm 				 := g_tyNtParamCurr.sMag1AWEngageProgNm;
	tylocalPneu.In.bExtSen 				 := g_tyDInput.bMag1WallEngageRS;
	tylocalPneu.In.bRetSen 				 := g_tyDInput.bMag1WallDisengageRS;
	tylocalPneu.In.tExtTO 				 := g_tyNtParamCurr.tMag1AWEngageExtTO;
	tylocalPneu.In.tRetTO 				 := g_tyNtParamCurr.tMag1AWEngageRetTO;
	tylocalPneu.In.ePneuSel				 := Pneu2Sen;

	IF g_tyStartUp.bRun = TRUE THEN
		tylocalPneu.In.eAct := g_tyOpsMagConvUL1MagAWEngageAct;
	ELSIF tylocalPneu.In.bManual = TRUE THEN
		tylocalPneu.In.eAct := g_tyUIMag1AWEngageAct;
	ELSE
		tylocalPneu.In.eAct := eAct;
	END_IF

END_ACTION
```

#### Act_OutputConfig.st
```iecst
ACTION Act_OutputConfig:
	// Output: Assign To Global For Independent Package Usage

	g_tyPneuMag1AWEngage := tylocalPneu.Out; // Change the Global Naming According to the Physical Hardware Module

END_ACTION
```

### Program Logical/Pneu/PneuMag2AWEngage (IEC) - 1.00.0 - NtPneu v5.00.0

#### Local.var
```iecst
(**)
VAR
	tylocalPneu : tyPneu;
END_VAR
(**)
VAR
	eAct : ePneuAction;
	udiStatus : UDINT := 0;
	bRstErr : BOOL;
	udiRstErrOld : UDINT;
	bInitialDone : BOOL;
	fbPneuNoSenExt : fbPneuNoSenExtChk;
	fbPneuNoSenRet : fbPneuNoSenRetChk;
	fbPneu2SenExt : fbPneuExtRetSenExtChk;
	fbPneu2SenRet : fbPneuExtRetSenRetChk;
	eStatOld : ePneuAction := PneuActIdle;
	bExtSen : BOOL;
	bRetSen : BOOL;
	bExtSafetySen : BOOL;
	bRetSafetySen : BOOL;
	udiModuleNum : UDINT := 2551;
END_VAR
```

#### Act_InputConfig.st
```iecst
ACTION Act_InputConfig:

	(* Always Change If Project Change *)

	//Pass Data To Link
	tylocalPneu.In.bSafetyRelaySig 	 	 := g_tyDInput.bSafetyRlySig;
	tylocalPneu.In.udiRstErr		 	 := g_tyRstErrOut.udiRstErr;
	tylocalPneu.In.bPrep 				 := g_tyNtParamCurr.bProjMagAWPrep;
	tylocalPneu.In.bDis 				 := g_tyMcParamCurr.bMagAWDis;
	tylocalPneu.In.bManual 				 := g_tyUIOut.bUIManualMod;
	tylocalPneu.In.bTwoCtrlIn 			 := g_tyNtParamCurr.bMag2AWEngageTwoCtrlIn;
	tylocalPneu.In.sProgNm 				 := g_tyNtParamCurr.sMag2AWEngageProgNm;
	tylocalPneu.In.bExtSen 				 := g_tyDInput.bMag2WallEngageRS;
	tylocalPneu.In.bRetSen 				 := g_tyDInput.bMag2WallDisengageRS;
	tylocalPneu.In.tExtTO 				 := g_tyNtParamCurr.tMag2AWEngageExtTO;
	tylocalPneu.In.tRetTO 				 := g_tyNtParamCurr.tMag2AWEngageRetTO;
	tylocalPneu.In.ePneuSel				 := Pneu2Sen;

	IF g_tyStartUp.bRun = TRUE THEN
		tylocalPneu.In.eAct := g_tyOpsMagConvUL2MagAWEngageAct;
	ELSIF tylocalPneu.In.bManual = TRUE THEN
		tylocalPneu.In.eAct := g_tyUIMag2AWEngageAct;
	ELSE
		tylocalPneu.In.eAct := eAct;
	END_IF

END_ACTION
```

#### Act_OutputConfig.st
```iecst
ACTION Act_OutputConfig:
	// Output: Assign To Global For Independent Package Usage

	g_tyPneuMag2AWEngage := tylocalPneu.Out; // Change the Global Naming According to the Physical Hardware Module

END_ACTION
```

### Program Logical/Pneu/PneuMag3AWEngage (IEC) - 1.00.0 - NtPneu v5.00.0

#### Act_InputConfig.st
```iecst
ACTION Act_InputConfig:

	(* Always Change If Project Change *)

	//Pass Data To Link
	tylocalPneu.In.bSafetyRelaySig 	 	 := g_tyDInput.bSafetyRlySig;
	tylocalPneu.In.udiRstErr		 	 := g_tyRstErrOut.udiRstErr;
	tylocalPneu.In.bPrep 				 := g_tyNtParamCurr.bProjMagAWPrep;
	tylocalPneu.In.bDis 				 := g_tyMcParamCurr.bMagAWDis;
	tylocalPneu.In.bManual 				 := g_tyUIOut.bUIManualMod;
	tylocalPneu.In.bTwoCtrlIn 			 := g_tyNtParamCurr.bMag3AWEngageTwoCtrlIn;
	tylocalPneu.In.sProgNm 				 := g_tyNtParamCurr.sMag3AWEngageProgNm;
	tylocalPneu.In.bExtSen 				 := g_tyDInput.bMag3WallEngageRS;
	tylocalPneu.In.bRetSen 				 := g_tyDInput.bMag3WallDisengageRS;
	tylocalPneu.In.tExtTO 				 := g_tyNtParamCurr.tMag3AWEngageExtTO;
	tylocalPneu.In.tRetTO 				 := g_tyNtParamCurr.tMag3AWEngageRetTO;
	tylocalPneu.In.ePneuSel				 := Pneu2Sen;

	IF g_tyStartUp.bRun = TRUE THEN
		tylocalPneu.In.eAct := g_tyOpsMagConvUL3MagAWEngageAct;
	ELSIF tylocalPneu.In.bManual = TRUE THEN
		tylocalPneu.In.eAct := g_tyUIMag3AWEngageAct;
	ELSE
		tylocalPneu.In.eAct := eAct;
	END_IF

END_ACTION
```

#### Act_Main.st
```iecst
ACTION Act_Main:

	IF tylocalPneu.In.bSafetyRelaySig = FALSE OR EDGEPOS(tylocalPneu.Out.eStatus = Error) THEN
		tylocalPneu.Out.bExtCtrl 	:= FALSE;
		tylocalPneu.Out.bRetCtrl 	:= FALSE;
		tylocalPneu.Out.bExtended	:= FALSE;
		tylocalPneu.Out.bRetracted  := FALSE;
	END_IF

	//Execution Action
	IF tylocalPneu.Out.eStatus <> Error THEN
		tylocalPneu.Out.eStat := tylocalPneu.In.eAct;
	END_IF

	//Transition State
	IF eStatOld <> tylocalPneu.Out.eStat THEN

		fbPneuNoSenExt(bEn := FALSE);
		fbPneuNoSenRet(bEn := FALSE);

		fbPneu2SenExt(bEn := FALSE);
		fbPneu2SenRet(bEn := FALSE);

		eStatOld	:= tylocalPneu.Out.eStat;

		tylocalPneu.Out.eStatus		:= Busy;
	END_IF

	//Main
	CASE tylocalPneu.Out.eStat OF

		PneuActIdle:
			tylocalPneu.Out.eStatus	:= Idle;

		PneuActSetAll:
			IF tylocalPneu.Out.eStatus = Idle OR tylocalPneu.Out.eStatus = Busy THEN

				fbPneuNoSenExt(bEn := FALSE);
				fbPneuNoSenRet(bEn := FALSE);

				fbPneu2SenExt(bEn := FALSE);
				fbPneu2SenRet(bEn := FALSE);

				tylocalPneu.Out.bExtCtrl	:= TRUE;
				tylocalPneu.Out.bRetCtrl	:= TRUE;

				tylocalPneu.Out.bExtended	:= FALSE;
				tylocalPneu.Out.bRetracted	:= FALSE;

				tylocalPneu.Out.eStatus	:= Done;

			END_IF

		PneuActRstAll:
			IF tylocalPneu.Out.eStatus = Idle OR tylocalPneu.Out.eStatus = Busy THEN

				fbPneuNoSenExt(bEn := FALSE);
				fbPneuNoSenRet(bEn := FALSE);

				fbPneu2SenExt(bEn := FALSE);
				fbPneu2SenRet(bEn := FALSE);

				tylocalPneu.Out.bExtCtrl	:= FALSE;
				tylocalPneu.Out.bRetCtrl	:= FALSE;

				tylocalPneu.Out.bExtended	:= FALSE;
				tylocalPneu.Out.bRetracted	:= FALSE;

				tylocalPneu.Out.eStatus	:= Done;

			END_IF

		PneuActSetExt:
			IF tylocalPneu.Out.eStatus = Idle OR tylocalPneu.Out.eStatus = Busy THEN

				fbPneuNoSenExt(bEn := FALSE);
				fbPneuNoSenRet(bEn := FALSE);

				fbPneu2SenExt(bEn := FALSE);
				fbPneu2SenRet(bEn := FALSE);

				tylocalPneu.Out.bExtCtrl	:= TRUE;
				tylocalPneu.Out.bRetCtrl	:= FALSE;

				tylocalPneu.Out.bExtended	:= TRUE;
				tylocalPneu.Out.bRetracted	:= FALSE;

				tylocalPneu.Out.eStatus	:= Done;

			END_IF

		PneuActSetRet:
			IF tylocalPneu.Out.eStatus = Idle OR tylocalPneu.Out.eStatus = Busy THEN

				//Reset
				fbPneuNoSenExt(bEn := FALSE);
				fbPneuNoSenRet(bEn := FALSE);

				fbPneu2SenExt(bEn := FALSE);
				fbPneu2SenRet(bEn := FALSE);

				tylocalPneu.Out.bExtCtrl	:= FALSE;
				tylocalPneu.Out.bRetCtrl	:= TRUE;

				tylocalPneu.Out.bExtended	:= FALSE;
				tylocalPneu.Out.bRetracted	:= TRUE;

				tylocalPneu.Out.eStatus	:= Done;

			END_IF

		PneuActExt:
			IF tylocalPneu.Out.eStatus = Idle OR tylocalPneu.Out.eStatus = Busy THEN

				tylocalPneu.Out.eStatus	:= Busy;

				tylocalPneu.Out.bExtCtrl	:= TRUE;
				tylocalPneu.Out.bRetCtrl	:= FALSE;

				CASE tylocalPneu.In.ePneuSel OF

					PneuNoSen: //Pneumatic Without Sen // 0
						fbPneuNoSenExt.bExtSafety	:= tylocalPneu.In.bExtSafetySen;
						fbPneuNoSenExt.tDlyTm		:= tylocalPneu.In.tExtDlyTm;
						fbPneuNoSenExt(bEn := TRUE);
					Pneu2Sen: //Pneumatic With 2 Sen // 3
						fbPneu2SenExt.bExtSen   	:= tylocalPneu.In.bExtSen;
						fbPneu2SenExt.bRetSen   	:= tylocalPneu.In.bRetSen;
						fbPneu2SenExt.bExtSafety	:= tylocalPneu.In.bExtSafetySen;
						fbPneu2SenExt.tTimeOut		:= tylocalPneu.In.tExtTO;
						fbPneu2SenExt(bEn := TRUE);
				END_CASE

				IF fbPneuNoSenExt.udiStatus = 0 OR
					fbPneu2SenExt.udiStatus = 0 THEN

					tylocalPneu.Out.bExtended	:= TRUE;
					tylocalPneu.Out.bRetracted	:= FALSE;
					tylocalPneu.Out.eStatus		:= Done;

				ELSIF (fbPneuNoSenExt.udiStatus > 0 AND fbPneuNoSenExt.udiStatus < 65534) OR
					(fbPneu2SenExt.udiStatus > 0 AND fbPneu2SenExt.udiStatus < 65534) THEN

					IF tylocalPneu.In.bTwoCtrlIn = TRUE THEN

						tylocalPneu.Out.bExtCtrl	:= FALSE;
						tylocalPneu.Out.bRetCtrl	:= FALSE;

					ELSE
						tylocalPneu.Out.bExtCtrl	:= FALSE;
						tylocalPneu.Out.bRetCtrl	:= TRUE;

					END_IF

					tylocalPneu.Out.bExtended	:= FALSE;
					tylocalPneu.Out.bRetracted	:= FALSE;

					tylocalPneu.Out.eStatus		:= Error;

					IF fbPneuNoSenExt.udiStatus = 1507 OR fbPneu2SenExt.udiStatus  = 1507 THEN
						udiStatus	:= 2401; //Safety Check Error While Extending
					ELSIF fbPneu2SenExt.udiStatus = 1503 THEN
						udiStatus	:= 2552;	//Extend Sensor On Checking Time Out While Extending
					ELSIF fbPneu2SenExt.udiStatus = 1506 THEN
						udiStatus	:= 2553; //Retract Sensor Off Checking Time Out While Extending
					ELSE
						IF tylocalPneu.In.ePneuSel = PneuNoSen THEN
							udiStatus	:= fbPneuNoSenExt.udiStatus;
						ELSE
							udiStatus	:= fbPneu2SenExt.udiStatus;
						END_IF
					END_IF
				END_IF

			END_IF

		PneuActRet:
			IF tylocalPneu.Out.eStatus = Idle OR tylocalPneu.Out.eStatus = Busy THEN

				tylocalPneu.Out.eStatus	:= Busy;

				tylocalPneu.Out.bExtCtrl	:= FALSE;
				tylocalPneu.Out.bRetCtrl	:= TRUE;

				CASE tylocalPneu.In.ePneuSel OF

					PneuNoSen: //Pneumatic Without Sen // 0
						fbPneuNoSenRet.bRetSafety	:= tylocalPneu.In.bRetSafetySen;
						fbPneuNoSenRet.tDlyTm		:= tylocalPneu.In.tRetDlyTm;
						fbPneuNoSenRet(bEn := TRUE);
					Pneu2Sen: //Pneumatic With 2 Sen // 3
						fbPneu2SenRet.bExtSen   	:= tylocalPneu.In.bExtSen;
						fbPneu2SenRet.bRetSen   	:= tylocalPneu.In.bRetSen;
						fbPneu2SenRet.bRetSafety	:= tylocalPneu.In.bRetSafetySen;
						fbPneu2SenRet.tTimeOut		:= tylocalPneu.In.tRetTO;
						fbPneu2SenRet(bEn := TRUE);
				END_CASE

				IF fbPneuNoSenRet.udiStatus = 0 OR
					fbPneu2SenRet.udiStatus = 0 THEN

					tylocalPneu.Out.bExtended	:= FALSE;
					tylocalPneu.Out.bRetracted	:= TRUE;
					tylocalPneu.Out.eStatus		:= Done;

				ELSIF (fbPneuNoSenRet.udiStatus > 0 AND fbPneuNoSenRet.udiStatus < 65534) OR
					(fbPneu2SenRet.udiStatus > 0 AND fbPneu2SenRet.udiStatus < 65534) THEN

					IF tylocalPneu.In.bTwoCtrlIn = TRUE THEN
						tylocalPneu.Out.bExtCtrl	:= FALSE;
						tylocalPneu.Out.bRetCtrl	:= FALSE;
					ELSE
						tylocalPneu.Out.bExtCtrl	:= TRUE;
						tylocalPneu.Out.bRetCtrl	:= FALSE;
					END_IF

					tylocalPneu.Out.bExtended	:= FALSE;
					tylocalPneu.Out.bRetracted	:= FALSE;

					tylocalPneu.Out.eStatus		:= Error;

					IF fbPneuNoSenRet.udiStatus = 1508 OR fbPneu2SenRet.udiStatus = 1508 THEN
						udiStatus	:= 2404;	//Safety Check Error While Retracting
					ELSIF fbPneu2SenRet.udiStatus = 1505 THEN
						udiStatus	:= 2555;	//Retract Sensor On Checking Time Out While Retracting
					ELSIF fbPneu2SenRet.udiStatus = 1504 THEN
						udiStatus	:= 2556;    //Extend Sensor Off Checking Time Out While Retracting
					ELSE
						IF tylocalPneu.In.ePneuSel = PneuNoSen THEN
							udiStatus	:= fbPneuNoSenRet.udiStatus;
						ELSE
							udiStatus	:= fbPneu2SenRet.udiStatus;
						END_IF
					END_IF
				END_IF

			END_IF

		ELSE
			IF tylocalPneu.Out.eStatus = Idle OR tylocalPneu.Out.eStatus = Busy THEN
				tylocalPneu.Out.eStatus	:= Done;
			END_IF

	END_CASE

	//background
	IF tylocalPneu.In.ePneuSel = Pneu2Sen THEN
		IF tylocalPneu.In.bExtSen = FALSE THEN
			tylocalPneu.Out.bExtended	:= FALSE;
		END_IF

		IF tylocalPneu.In.bRetSen = FALSE THEN
			tylocalPneu.Out.bRetracted	:= FALSE;
		END_IF
	END_IFs

END_ACTION
```

#### Act_OutputConfig.st
```iecst
ACTION Act_OutputConfig:
	// Output: Assign To Global For Independent Package Usage

	g_tyPneuMag3AWEngage := tylocalPneu.Out; // Change the Global Naming According to the Physical Hardware Module

END_ACTION
```

### Pneu2SenMag1AWEngage.var - not listed in the package file held
```iecst
(*2019-03-25*)
(**)
(*Action & State & Status*)
VAR
	p_Pneu2SMag1AWEngageStat : UDINT;
	p_Pneu2SMag1AWEngageStatus : UDINT;
	p_Pneu2SMag1AWEngageStatTxt : UDINT;
END_VAR
(**)
(*Alarm*)
VAR
	p_Pneu2SMag1AWEngageAlmData : UDINT;
END_VAR
(**)
(*Output*)
VAR
	p_Pneu2SMag1AWEngageExtCtrl : UDINT;
	p_Pneu2SMag1AWEngageRetCtrl : UDINT;
	p_Pneu2SMag1AWEngageTwoCtrlOut : UDINT;
	p_Pneu2SMag1AWEngageExtended : UDINT;
	p_Pneu2SMag1AWEngageRetracted : UDINT;
END_VAR
```

### Pneu2SenMag1SafetyBar.var - not listed in the package file held
```iecst
(*2019-03-25*)
(**)
(*Action & State & Status*)
VAR
	p_Pneu2SMag1SafetyBarStat : UDINT;
	p_Pneu2SMag1SafetyBarStatus : UDINT;
	p_Pneu2SMag1SafetyBarStatTxt : UDINT;
END_VAR
(**)
(*Alarm*)
VAR
	p_Pneu2SMag1SafetyBarAlmData : UDINT;
END_VAR
(**)
(*Output*)
VAR
	p_Pneu2SMag1SafetyBarExtCtrl : UDINT;
	p_Pneu2SMag1SafetyBarRetCtrl : UDINT;
	p_Pneu2SMag1SafetyBarTwoCtrlOut : UDINT;
	p_Pneu2SMag1SafetyBarExtended : UDINT;
	p_Pneu2SMag1SafetyBarRetracted : UDINT;
END_VAR
```

### Pneu2SenMag2AWEngage.var - not listed in the package file held
```iecst
(*2019-03-25*)
(**)
(*Action & State & Status*)
VAR
	p_Pneu2SMag2AWEngageStat : UDINT;
	p_Pneu2SMag2AWEngageStatus : UDINT;
	p_Pneu2SMag2AWEngageStatTxt : UDINT;
END_VAR
(**)
(*Alarm*)
VAR
	p_Pneu2SMag2AWEngageAlmData : UDINT;
END_VAR
(**)
(*Output*)
VAR
	p_Pneu2SMag2AWEngageExtCtrl : UDINT;
	p_Pneu2SMag2AWEngageRetCtrl : UDINT;
	p_Pneu2SMag2AWEngageTwoCtrlOut : UDINT;
	p_Pneu2SMag2AWEngageExtended : UDINT;
	p_Pneu2SMag2AWEngageRetracted : UDINT;
END_VAR
```

### Pneu2SenMag2SafetyBar.var - not listed in the package file held
```iecst
(*2019-03-25*)
(**)
(*Action & State & Status*)
VAR
	p_Pneu2SMag2SafetyBarStat : UDINT;
	p_Pneu2SMag2SafetyBarStatus : UDINT;
	p_Pneu2SMag2SafetyBarStatTxt : UDINT;
END_VAR
(**)
(*Alarm*)
VAR
	p_Pneu2SMag2SafetyBarAlmData : UDINT;
END_VAR
(**)
(*Output*)
VAR
	p_Pneu2SMag2SafetyBarExtCtrl : UDINT;
	p_Pneu2SMag2SafetyBarRetCtrl : UDINT;
	p_Pneu2SMag2SafetyBarTwoCtrlOut : UDINT;
	p_Pneu2SMag2SafetyBarExtended : UDINT;
	p_Pneu2SMag2SafetyBarRetracted : UDINT;
END_VAR
```

### Pneu2SenMag3AWEngage.var - not listed in the package file held
```iecst
(*2019-03-25*)
(**)
(*Action & State & Status*)
VAR
	p_Pneu2SMag3AWEngageStat : UDINT;
	p_Pneu2SMag3AWEngageStatus : UDINT;
	p_Pneu2SMag3AWEngageStatTxt : UDINT;
END_VAR
(**)
(*Alarm*)
VAR
	p_Pneu2SMag3AWEngageAlmData : UDINT;
END_VAR
(**)
(*Output*)
VAR
	p_Pneu2SMag3AWEngageExtCtrl : UDINT;
	p_Pneu2SMag3AWEngageRetCtrl : UDINT;
	p_Pneu2SMag3AWEngageTwoCtrlOut : UDINT;
	p_Pneu2SMag3AWEngageExtended : UDINT;
	p_Pneu2SMag3AWEngageRetracted : UDINT;
END_VAR
```

### Pneu2SenMag3SafetyBar.var - not listed in the package file held
```iecst
(*2019-03-25*)
(**)
(*Action & State & Status*)
VAR
	p_Pneu2SMag3SafetyBarStat : UDINT;
	p_Pneu2SMag3SafetyBarStatus : UDINT;
	p_Pneu2SMag3SafetyBarStatTxt : UDINT;
END_VAR
(**)
(*Alarm*)
VAR
	p_Pneu2SMag3SafetyBarAlmData : UDINT;
END_VAR
(**)
(*Output*)
VAR
	p_Pneu2SMag3SafetyBarExtCtrl : UDINT;
	p_Pneu2SMag3SafetyBarRetCtrl : UDINT;
	p_Pneu2SMag3SafetyBarTwoCtrlOut : UDINT;
	p_Pneu2SMag3SafetyBarExtended : UDINT;
	p_Pneu2SMag3SafetyBarRetracted : UDINT;
END_VAR
```

### Pneu2SenOutShutter2.var - not listed in the package file held
```iecst
(*2019-03-25*)
(**)
(*Action & State & Status*)
VAR
	p_Pneu2SenOutShutterStat2 : UDINT;
	p_Pneu2SenOutShutterStatus2 : UDINT;
	p_Pneu2SenOutShutterStatTxt2 : UDINT;
END_VAR
(**)
(*Alarm*)
VAR
	p_Pneu2SenOutShutterAlmData2 : UDINT;
END_VAR
(**)
(*Output*)
VAR
	p_Pneu2SenOutShutterExtCtrl2 : UDINT;
	p_Pneu2SenOutShutterRetCtrl2 : UDINT;
	p_Pneu2SenOutShutterTwoCtrlOut2 : UDINT;
	p_Pneu2SenOutShutterExtended2 : UDINT;
	p_Pneu2SenOutShutterRetracted2 : UDINT;
END_VAR
```

### Pneu2SenOutShutter3.var - not listed in the package file held
```iecst
(*2019-03-25*)
(**)
(*Action & State & Status*)
VAR
	p_Pneu2SenOutShutterStat3 : UDINT;
	p_Pneu2SenOutShutterStatus3 : UDINT;
	p_Pneu2SenOutShutterStatTxt3 : UDINT;
END_VAR
(**)
(*Alarm*)
VAR
	p_Pneu2SenOutShutterAlmData3 : UDINT;
END_VAR
(**)
(*Output*)
VAR
	p_Pneu2SenOutShutterExtCtrl3 : UDINT;
	p_Pneu2SenOutShutterRetCtrl3 : UDINT;
	p_Pneu2SenOutShutterTwoCtrlOut3 : UDINT;
	p_Pneu2SenOutShutterExtended3 : UDINT;
	p_Pneu2SenOutShutterRetracted3 : UDINT;
END_VAR
```

### Pneu2SenSelClamp1.var - not listed in the package file held
```iecst
(*2019-03-25*)
(**)
(*Action & State & Status*)
VAR
	p_PneuNoSenSelClamp1Stat : UDINT;
	p_PneuNoSenSelClamp1Status : UDINT;
	p_PneuNoSenSelClamp1StatTxt : UDINT;
END_VAR
(**)
(*Alarm*)
VAR
	p_PneuNoSenSelClamp1AlmData : UDINT;
END_VAR
(**)
(*Output*)
VAR
	p_PneuNoSenSelClamp1ExtCtrl : UDINT;
	p_PneuNoSenSelClamp1RetCtrl : UDINT;
	p_PneuNoSenSelClamp1TwoCtrlOut : UDINT;
	p_PneuNoSenSelClamp1Extended : UDINT;
	p_PneuNoSenSelClamp1Retracted : UDINT;
END_VAR
```

### Pneu2SenSelClamp2.var - not listed in the package file held
```iecst
(*2029-03-25*)
(**)
(*Action & State & Status*)
VAR
	p_PneuNoSenSelClamp2Stat : UDINT;
	p_PneuNoSenSelClamp2Status : UDINT;
	p_PneuNoSenSelClamp2StatTxt : UDINT;
END_VAR
(**)
(*Alarm*)
VAR
	p_PneuNoSenSelClamp2AlmData : UDINT;
END_VAR
(**)
(*Output*)
VAR
	p_PneuNoSenSelClamp2ExtCtrl : UDINT;
	p_PneuNoSenSelClamp2RetCtrl : UDINT;
	p_PneuNoSenSelClamp2TwoCtrlOut : UDINT;
	p_PneuNoSenSelClamp2Extended : UDINT;
	p_PneuNoSenSelClamp2Retracted : UDINT;
END_VAR
```

### Pneu2SenSelClamp3.var - not listed in the package file held
```iecst
(*2039-03-25*)
(**)
(*Action & State & Status*)
VAR
	p_PneuNoSenSelClamp3Stat : UDINT;
	p_PneuNoSenSelClamp3Status : UDINT;
	p_PneuNoSenSelClamp3StatTxt : UDINT;
END_VAR
(**)
(*Alarm*)
VAR
	p_PneuNoSenSelClamp3AlmData : UDINT;
END_VAR
(**)
(*Output*)
VAR
	p_PneuNoSenSelClamp3ExtCtrl : UDINT;
	p_PneuNoSenSelClamp3RetCtrl : UDINT;
	p_PneuNoSenSelClamp3TwoCtrlOut : UDINT;
	p_PneuNoSenSelClamp3Extended : UDINT;
	p_PneuNoSenSelClamp3Retracted : UDINT;
END_VAR
```

### PneuNoSenInletStopper.var - not listed in the package file held
```iecst
(*2019-03-25*)
(**)
(*Action & State & Status*)
VAR
	p_InletStopperStat : UDINT;
	p_InletStopperStatus : UDINT;
	p_InletStopperStatTxt : UDINT;
END_VAR
(**)
(*Alarm*)
VAR
	p_InletStopperAlmData : UDINT;
END_VAR
(**)
(*Output*)
VAR
	p_InletStopperExtCtrl : UDINT;
	p_InletStopperRetCtrl : UDINT;
	p_InletStopperTwoCtrlOut : UDINT;
	p_InletStopperExtended : UDINT;
	p_InletStopperRetracted : UDINT;
END_VAR
```

### PneuNoSenStopperA.var - not listed in the package file held
```iecst
(*2019-03-25*)
(**)
(*Action & State & Status*)
VAR
	p_PneuNoSenStopperAStat : UDINT;
	p_PneuNoSenStopperAStatus : UDINT;
	p_PneuNoSenStopperAStatTxt : UDINT;
END_VAR
(**)
(*Alarm*)
VAR
	p_PneuNoSenStopperAAlmData : UDINT;
END_VAR
(**)
(*Output*)
VAR
	p_PneuNoSenStopperAExtCtrl : UDINT;
	p_PneuNoSenStopperARetCtrl : UDINT;
	p_PneuNoSenStopperATwoCtrlOut : UDINT;
	p_PneuNoSenStopperAExtended : UDINT;
	p_PneuNoSenStopperARetracted : UDINT;
END_VAR
```

### PneuNoSenStopperB.var - not listed in the package file held
```iecst
(*2019-03-25*)
(**)
(*Action & State & Status*)
VAR
	p_PneuNoSenStopperBStat : UDINT;
	p_PneuNoSenStopperBStatus : UDINT;
	p_PneuNoSenStopperBStatTxt : UDINT;
END_VAR
(**)
(*Alarm*)
VAR
	p_PneuNoSenStopperBAlmData : UDINT;
END_VAR
(**)
(*Output*)
VAR
	p_PneuNoSenStopperBExtCtrl : UDINT;
	p_PneuNoSenStopperBRetCtrl : UDINT;
	p_PneuNoSenStopperBTwoCtrlOut : UDINT;
	p_PneuNoSenStopperBExtended : UDINT;
	p_PneuNoSenStopperBRetracted : UDINT;
END_VAR
```

### PneuNoSenStopperC.var - not listed in the package file held
```iecst
(*2019-03-25*)
(**)
(*Action & State & Status*)
VAR
	p_PneuNoSenStopperCStat : UDINT;
	p_PneuNoSenStopperCStatus : UDINT;
	p_PneuNoSenStopperCStatTxt : UDINT;
END_VAR
(**)
(*Alarm*)
VAR
	p_PneuNoSenStopperCAlmData : UDINT;
END_VAR
(**)
(*Output*)
VAR
	p_PneuNoSenStopperCExtCtrl : UDINT;
	p_PneuNoSenStopperCRetCtrl : UDINT;
	p_PneuNoSenStopperCTwoCtrlOut : UDINT;
	p_PneuNoSenStopperCExtended : UDINT;
	p_PneuNoSenStopperCRetracted : UDINT;
END_VAR
```

### PneuNoSenTopEntStpr.var - Change By Project
```iecst
(*2019-03-25*)
(**)
(*Action & State & Status*)
VAR
	p_PneuNoSenTopEntStprStat : UDINT;
	p_PneuNoSenTopEntStprStatus : UDINT;
	p_PneuNoSenTopEntStprStatTxt : UDINT;
END_VAR
(**)
(*Alarm*)
VAR
	p_PneuNoSenTopEntStprAlmData : UDINT;
END_VAR
(**)
(*Output*)
VAR
	p_PneuNoSenTopEntStprExtCtrl : UDINT;
	p_PneuNoSenTopEntStprRetCtrl : UDINT;
	p_PneuNoSenTopEntStprTwoCtrlOut : UDINT;
	p_PneuNoSenTopEntStprExtended : UDINT;
	p_PneuNoSenTopEntStprRetracted : UDINT;
END_VAR
```

### Program Logical/Pneu/MagConv_Stopper/PneuNoSenTopEntStpr (IEC) - 1.00.0 - NtPneu v5.00.0

#### Act_InitGlobal.st
```iecst
(** 2019-04-09 **)
ACTION Act_InitGlobal:

	(* Always Change If Project Change *)

	//Pass Data To Link
	p_bLinkOpsRun ACCESS p_OpsRun;

	p_bLinkDISafetyRlySig ACCESS p_DISafetyRlySig;

	//Pass Data To Internal Use
	p_udiRstErr ACCESS p_RstErrReset;
	p_bPrep ACCESS p_NtParamProjTopEntStprPrep;
//	p_bDis ACCESS p_McParamTopEntStprDis;
	p_bManual ACCESS p_UIMnlMod;
	p_bTwoCtrlIn ACCESS p_NtParamTopEntStprTwoCtrlIn;
	p_sProgNm ACCESS p_NtParamTopEntStprProgNm;
	p_tExtDlyTm ACCESS p_NtParamTopEntStprExtDlyTm;
	p_tRetDlyTm ACCESS p_NtParamTopEntStprRetDlyTm;
	p_bNtSettingsLoadDone ACCESS p_StartupNtSettingsLoadDone;
	p_bPrep ACCESS p_NtParamProjMagConvLane1Prep;
	(* Always Change If Project Change *)

END_ACTION
```

#### Act_LinkAction.st
```iecst
(** 2019-04-09 **)
ACTION Act_LinkAction:

	IF p_bLinkOpsRun = TRUE AND p_OpsMagConvStprTopEntAct <> 0 THEN
		p_eAct ACCESS p_OpsMagConvStprTopEntAct;
	ELSIF p_bManual = TRUE THEN
		p_eAct ACCESS p_UIStopper1Act;
	ELSE
		p_eAct ACCESS ADR(eAct);
	END_IF

END_ACTION
```

#### Init.st
```iecst
(** 2019-03-25 **)
PROGRAM _INIT

	(* Always Change If Project Change *)

	//Pass Address To Global Address For External Use
	//Action, State & Status
	p_PneuNoSenTopEntStprStat			:= ADR(eStat);
	p_PneuNoSenTopEntStprStatus			:= ADR(eStatus);
	p_PneuNoSenTopEntStprStatTxt		:= ADR(sStatTxt);

	//Alarm
	p_PneuNoSenTopEntStprAlmData		:= ADR(tyAlmData);

	//Output
	p_PneuNoSenTopEntStprExtCtrl		:= ADR(bExtCtrl);
	p_PneuNoSenTopEntStprRetCtrl		:= ADR(bRetCtrl);
	p_PneuNoSenTopEntStprTwoCtrlOut		:= ADR(bTwoCtrlOut);
	p_PneuNoSenTopEntStprExtended		:= ADR(bExtended);
	p_PneuNoSenTopEntStprRetracted		:= ADR(bRetracted);

	(* Always Change If Project Change *)

END_PROGRAM
```

### PneuNoSenTopMidStpr.var - Change By Project
```iecst
(*2019-03-25*)
(**)
(*Action & State & Status*)
VAR
	p_PneuNoSenTopMidStprStat : UDINT;
	p_PneuNoSenTopMidStprStatus : UDINT;
	p_PneuNoSenTopMidStprStatTxt : UDINT;
END_VAR
(**)
(*Alarm*)
VAR
	p_PneuNoSenTopMidStprAlmData : UDINT;
END_VAR
(**)
(*Output*)
VAR
	p_PneuNoSenTopMidStprExtCtrl : UDINT;
	p_PneuNoSenTopMidStprRetCtrl : UDINT;
	p_PneuNoSenTopMidStprTwoCtrlOut : UDINT;
	p_PneuNoSenTopMidStprExtended : UDINT;
	p_PneuNoSenTopMidStprRetracted : UDINT;
END_VAR
```

### Program Logical/Pneu/MagConv_Stopper/PneuNoSenTopMidStpr (IEC) - 1.00.0 - NtPneu v5.00.0

#### Act_InitGlobal.st
```iecst
(** 2019-04-09 **)
ACTION Act_InitGlobal:

	(* Always Change If Project Change *)

	//Pass Data To Link
	p_bLinkOpsRun ACCESS p_OpsRun;

	p_bLinkDISafetyRlySig ACCESS p_DISafetyRlySig;

	//Pass Data To Internal Use
	p_udiRstErr ACCESS p_RstErrReset;
	p_bPrep ACCESS p_NtParamProjTopMidStprPrep;
//	p_bDis ACCESS p_McParamTopMidStprDis;
	p_bManual ACCESS p_UIMnlMod;
	p_bTwoCtrlIn ACCESS p_NtParamTopMidStprTwoCtrlIn;
	p_sProgNm ACCESS p_NtParamTopMidStprProgNm;
	p_tExtDlyTm ACCESS p_NtParamTopMidStprExtDlyTm;
	p_tRetDlyTm ACCESS p_NtParamTopMidStprRetDlyTm;
	p_bNtSettingsLoadDone ACCESS p_StartupNtSettingsLoadDone;
	p_bPrep ACCESS p_NtParamProjMagConvLane1Prep;
	(* Always Change If Project Change *)

END_ACTION
```

#### Act_LinkAction.st
```iecst
(** 2019-04-09 **)
ACTION Act_LinkAction:

	IF p_bLinkOpsRun = TRUE AND p_OpsMagConvStprTopMidAct <> 0 THEN
//		p_eAct ACCESS p_OpsTravLifULStopperAct1;
		p_eAct ACCESS p_OpsMagConvStprTopMidAct;
	ELSIF p_bManual = TRUE THEN
		p_eAct ACCESS p_UIStopper2Act;
	ELSE
		p_eAct ACCESS ADR(eAct);
	END_IF

END_ACTION
```

#### Init.st
```iecst
(** 2019-03-25 **)
PROGRAM _INIT

	(* Always Change If Project Change *)

	//Pass Address To Global Address For External Use
	//Action, State & Status
	p_PneuNoSenTopMidStprStat			:= ADR(eStat);
	p_PneuNoSenTopMidStprStatus			:= ADR(eStatus);
	p_PneuNoSenTopMidStprStatTxt		:= ADR(sStatTxt);

	//Alarm
	p_PneuNoSenTopMidStprAlmData		:= ADR(tyAlmData);

	//Output
	p_PneuNoSenTopMidStprExtCtrl		:= ADR(bExtCtrl);
	p_PneuNoSenTopMidStprRetCtrl		:= ADR(bRetCtrl);
	p_PneuNoSenTopMidStprTwoCtrlOut		:= ADR(bTwoCtrlOut);
	p_PneuNoSenTopMidStprExtended		:= ADR(bExtended);
	p_PneuNoSenTopMidStprRetracted		:= ADR(bRetracted);

	(* Always Change If Project Change *)

END_PROGRAM
```

### PneuNoSenTopExtStpr.var - Change By Project
```iecst
(*2019-03-25*)
(**)
(*Action & State & Status*)
VAR
	p_PneuNoSenTopExtStprStat : UDINT;
	p_PneuNoSenTopExtStprStatus : UDINT;
	p_PneuNoSenTopExtStprStatTxt : UDINT;
END_VAR
(**)
(*Alarm*)
VAR
	p_PneuNoSenTopExtStprAlmData : UDINT;
END_VAR
(**)
(*Output*)
VAR
	p_PneuNoSenTopExtStprExtCtrl : UDINT;
	p_PneuNoSenTopExtStprRetCtrl : UDINT;
	p_PneuNoSenTopExtStprTwoCtrlOut : UDINT;
	p_PneuNoSenTopExtStprExtended : UDINT;
	p_PneuNoSenTopExtStprRetracted : UDINT;
END_VAR
```

### Program Logical/Pneu/MagConv_Stopper/PneuNoSenTopExtStpr (IEC) - 1.00.0 - NtPneu v5.00.0

#### Act_InitGlobal.st
```iecst
(** 2019-04-09 **)
ACTION Act_InitGlobal:

	(* Always Change If Project Change *)

	//Pass Data To Link
	p_bLinkOpsRun ACCESS p_OpsRun;

	p_bLinkDISafetyRlySig ACCESS p_DISafetyRlySig;

	//Pass Data To Internal Use
	p_udiRstErr ACCESS p_RstErrReset;
	p_bPrep ACCESS p_NtParamProjTopExtStprPrep;
//	p_bDis ACCESS p_McParamTopExtStprDis;
	p_bManual ACCESS p_UIMnlMod;
	p_bTwoCtrlIn ACCESS p_NtParamTopExtStprTwoCtrlIn;
	p_sProgNm ACCESS p_NtParamTopExtStprProgNm;
	p_tExtDlyTm ACCESS p_NtParamTopExtStprExtDlyTm;
	p_tRetDlyTm ACCESS p_NtParamTopExtStprRetDlyTm;
	p_bNtSettingsLoadDone ACCESS p_StartupNtSettingsLoadDone;
	p_bPrep ACCESS p_NtParamProjMagConvLane1Prep;
	(* Always Change If Project Change *)

END_ACTION
```

#### Act_LinkAction.st
```iecst
(** 2019-04-09 **)
ACTION Act_LinkAction:

	IF p_bLinkOpsRun = TRUE AND p_OpsMagConvStprTopExitAct<> 0 THEN
		//	p_eAct ACCESS p_OpsTravLifULStopperAct1;
		p_eAct ACCESS p_OpsMagConvStprTopExitAct;
	ELSIF p_bManual = TRUE THEN
		p_eAct ACCESS p_UIStopper3Act;
	ELSE
		p_eAct ACCESS ADR(eAct);
	END_IF

END_ACTION
```

#### Init.st
```iecst
(** 2019-03-25 **)
PROGRAM _INIT

	(* Always Change If Project Change *)

	//Pass Address To Global Address For External Use
	//Action, State & Status
	p_PneuNoSenTopExtStprStat			:= ADR(eStat);
	p_PneuNoSenTopExtStprStatus			:= ADR(eStatus);
	p_PneuNoSenTopExtStprStatTxt		:= ADR(sStatTxt);

	//Alarm
	p_PneuNoSenTopExtStprAlmData		:= ADR(tyAlmData);

	//Output
	p_PneuNoSenTopExtStprExtCtrl		:= ADR(bExtCtrl);
	p_PneuNoSenTopExtStprRetCtrl		:= ADR(bRetCtrl);
	p_PneuNoSenTopExtStprTwoCtrlOut		:= ADR(bTwoCtrlOut);
	p_PneuNoSenTopExtStprExtended		:= ADR(bExtended);
	p_PneuNoSenTopExtStprRetracted		:= ADR(bRetracted);

	(* Always Change If Project Change *)

END_PROGRAM
```

### PneuNoSenBtmMidStpr.var - Change By Project
```iecst
(*2019-03-25*)
(**)
(*Action & State & Status*)
VAR
	p_PneuNoSenBtmMidStprStat : UDINT;
	p_PneuNoSenBtmMidStprStatus : UDINT;
	p_PneuNoSenBtmMidStprStatTxt : UDINT;
END_VAR
(**)
(*Alarm*)
VAR
	p_PneuNoSenBtmMidStprAlmData : UDINT;
END_VAR
(**)
(*Output*)
VAR
	p_PneuNoSenBtmMidStprExtCtrl : UDINT;
	p_PneuNoSenBtmMidStprRetCtrl : UDINT;
	p_PneuNoSenBtmMidStprTwoCtrlOut : UDINT;
	p_PneuNoSenBtmMidStprExtended : UDINT;
	p_PneuNoSenBtmMidStprRetracted : UDINT;
END_VAR
```

### Program Logical/Pneu/MagConv_Stopper/PneuNoSenBtmMidStpr (IEC) - 1.00.0 - NtPneu v5.00.0

#### Act_InitGlobal.st
```iecst
(** 2019-04-09 **)
ACTION Act_InitGlobal:

	(* Always Change If Project Change *)

	//Pass Data To Link
	p_bLinkOpsRun ACCESS p_OpsRun;

	p_bLinkDISafetyRlySig ACCESS p_DISafetyRlySig;

	//Pass Data To Internal Use
	p_udiRstErr ACCESS p_RstErrReset;
	p_bPrep ACCESS p_NtParamProjBtmMidStprPrep;
//	p_bDis ACCESS p_McParamBtmMidStprDis;
	p_bManual ACCESS p_UIMnlMod;
	p_bTwoCtrlIn ACCESS p_NtParamBtmMidStprTwoCtrlIn;
	p_sProgNm ACCESS p_NtParamBtmMidStprProgNm;
	p_tExtDlyTm ACCESS p_NtParamBtmMidStprExtDlyTm;
	p_tRetDlyTm ACCESS p_NtParamBtmMidStprRetDlyTm;
	p_bNtSettingsLoadDone ACCESS p_StartupNtSettingsLoadDone;
	p_bPrep ACCESS p_NtParamProjMagConvLane1Prep;
	(* Always Change If Project Change *)

END_ACTION
```

#### Act_LinkAction.st
```iecst
(** 2019-04-09 **)
ACTION Act_LinkAction:

	IF p_bLinkOpsRun = TRUE AND p_OpsMagConvStprBtmMidAct <> 0 THEN
//		p_eAct ACCESS p_OpsTravLifULStopperAct1;
		p_eAct ACCESS p_OpsMagConvStprBtmMidAct;
	ELSIF p_bManual = TRUE THEN
		p_eAct ACCESS p_UIStopper4Act;
	ELSE
		p_eAct ACCESS ADR(eAct);
	END_IF

END_ACTION
```

#### Init.st
```iecst
(** 2019-03-25 **)
PROGRAM _INIT

	(* Always Change If Project Change *)

	//Pass Address To Global Address For External Use
	//Action, State & Status
	p_PneuNoSenBtmMidStprStat			:= ADR(eStat);
	p_PneuNoSenBtmMidStprStatus			:= ADR(eStatus);
	p_PneuNoSenBtmMidStprStatTxt		:= ADR(sStatTxt);

	//Alarm
	p_PneuNoSenBtmMidStprAlmData		:= ADR(tyAlmData);

	//Output
	p_PneuNoSenBtmMidStprExtCtrl		:= ADR(bExtCtrl);
	p_PneuNoSenBtmMidStprRetCtrl		:= ADR(bRetCtrl);
	p_PneuNoSenBtmMidStprTwoCtrlOut		:= ADR(bTwoCtrlOut);
	p_PneuNoSenBtmMidStprExtended		:= ADR(bExtended);
	p_PneuNoSenBtmMidStprRetracted		:= ADR(bRetracted);

	(* Always Change If Project Change *)

END_PROGRAM
```

### PneuNoSenBtmExtStpr.var - Change By Project
```iecst
(*2019-03-25*)
(**)
(*Action & State & Status*)
VAR
	p_PneuNoSenBtmExtStprStat : UDINT;
	p_PneuNoSenBtmExtStprStatus : UDINT;
	p_PneuNoSenBtmExtStprStatTxt : UDINT;
END_VAR
(**)
(*Alarm*)
VAR
	p_PneuNoSenBtmExtStprAlmData : UDINT;
END_VAR
(**)
(*Output*)
VAR
	p_PneuNoSenBtmExtStprExtCtrl : UDINT;
	p_PneuNoSenBtmExtStprRetCtrl : UDINT;
	p_PneuNoSenBtmExtStprTwoCtrlOut : UDINT;
	p_PneuNoSenBtmExtStprExtended : UDINT;
	p_PneuNoSenBtmExtStprRetracted : UDINT;
END_VAR
```

### Program Logical/Pneu/MagConv_Stopper/PneuNoSenBtmExtStpr (IEC) - 1.00.0 - NtPneu v5.00.0

#### Act_InitGlobal.st
```iecst
(** 2019-04-09 **)
ACTION Act_InitGlobal:

	(* Always Change If Project Change *)

	//Pass Data To Link
	p_bLinkOpsRun ACCESS p_OpsRun;

	p_bLinkDISafetyRlySig ACCESS p_DISafetyRlySig;

	//Pass Data To Internal Use
	p_udiRstErr ACCESS p_RstErrReset;
	p_bPrep ACCESS p_NtParamProjBtmExtStprPrep;
//	p_bDis ACCESS p_McParamBtmExtStprDis;
	p_bManual ACCESS p_UIMnlMod;
	p_bTwoCtrlIn ACCESS p_NtParamBtmExtStprTwoCtrlIn;
	p_sProgNm ACCESS p_NtParamBtmExtStprProgNm;
	p_tExtDlyTm ACCESS p_NtParamBtmExtStprExtDlyTm;
	p_tRetDlyTm ACCESS p_NtParamBtmExtStprRetDlyTm;
	p_bNtSettingsLoadDone ACCESS p_StartupNtSettingsLoadDone;
	p_bPrep ACCESS p_NtParamProjMagConvLane1Prep;
	(* Always Change If Project Change *)

END_ACTION
```

#### Act_LinkAction.st
```iecst
(** 2019-04-09 **)
ACTION Act_LinkAction:

	IF p_bLinkOpsRun = TRUE AND p_OpsMagConvStprBtmExitAct <> 0 THEN
//		p_eAct ACCESS p_OpsTravLifULStopperAct1;
		p_eAct ACCESS 	p_OpsMagConvStprBtmExitAct;
	ELSIF p_bManual = TRUE THEN
		p_eAct ACCESS p_UIStopper5Act;
	ELSE
		p_eAct ACCESS ADR(eAct);
	END_IF

END_ACTION
```

#### Init.st
```iecst
(** 2019-03-25 **)
PROGRAM _INIT

	(* Always Change If Project Change *)

	//Pass Address To Global Address For External Use
	//Action, State & Status
	p_PneuNoSenBtmExtStprStat			:= ADR(eStat);
	p_PneuNoSenBtmExtStprStatus			:= ADR(eStatus);
	p_PneuNoSenBtmExtStprStatTxt		:= ADR(sStatTxt);

	//Alarm
	p_PneuNoSenBtmExtStprAlmData		:= ADR(tyAlmData);

	//Output
	p_PneuNoSenBtmExtStprExtCtrl		:= ADR(bExtCtrl);
	p_PneuNoSenBtmExtStprRetCtrl		:= ADR(bRetCtrl);
	p_PneuNoSenBtmExtStprTwoCtrlOut		:= ADR(bTwoCtrlOut);
	p_PneuNoSenBtmExtStprExtended		:= ADR(bExtended);
	p_PneuNoSenBtmExtStprRetracted		:= ADR(bRetracted);

	(* Always Change If Project Change *)

END_PROGRAM
```

### PneuNoSenTopEntStpr2.var - Change By Project
```iecst
(*2019-03-25*)
(**)
(*Action & State & Status*)
VAR
	p_PneuNoSenTopEntStpr2Stat : UDINT;
	p_PneuNoSenTopEntStpr2Status : UDINT;
	p_PneuNoSenTopEntStpr2StatTxt : UDINT;
END_VAR
(**)
(*Alarm*)
VAR
	p_PneuNoSenTopEntStpr2AlmData : UDINT;
END_VAR
(**)
(*Output*)
VAR
	p_PneuNoSenTopEntStpr2ExtCtrl : UDINT;
	p_PneuNoSenTopEntStpr2RetCtrl : UDINT;
	p_PneuNoSenTopEntStpr2TwoCtrlOut : UDINT;
	p_PneuNoSenTopEntStpr2Extended : UDINT;
	p_PneuNoSenTopEntStpr2Retracted : UDINT;
END_VAR
```

### Program Logical/Pneu/MagConv_Stopper/PneuNoSenTopEntStpr2 (IEC) - 1.00.0 - NtPneu v5.00.0

#### Act_InitGlobal.st
```iecst
(** 2019-04-09 **)
ACTION Act_InitGlobal:

	(* Always Change If Project Change *)

	//Pass Data To Link
	p_bLinkOpsRun ACCESS p_OpsRun;

	p_bLinkDISafetyRlySig ACCESS p_DISafetyRlySig;

	//Pass Data To Internal Use
	p_udiRstErr ACCESS p_RstErrReset;
	p_bPrep ACCESS p_NtParamProjTopEntStprPrep2;
//	p_bDis ACCESS p_McParamTopEntStpr2Dis;
	p_bManual ACCESS p_UIMnlMod;
	p_bTwoCtrlIn ACCESS p_NtParamTopEntStprTwoCtrlIn2;
	p_sProgNm ACCESS p_NtParamTopEntStprProgNm2;
	p_tExtDlyTm ACCESS p_NtParamTopEntStprExtDlyTm2;
	p_tRetDlyTm ACCESS p_NtParamTopEntStprRetDlyTm2;
	p_bNtSettingsLoadDone ACCESS p_StartupNtSettingsLoadDone;
	p_bPrep ACCESS p_NtParamProjMagConvLane2Prep;
	(* Always Change If Project Change *)

END_ACTION
```

#### Act_LinkAction.st
```iecst
(** 2019-04-09 **)
ACTION Act_LinkAction:

	IF p_bLinkOpsRun = TRUE AND p_OpsMagConv2StprTopEntAct <> 0 THEN
		p_eAct ACCESS p_OpsMagConv2StprTopEntAct;
	ELSIF p_bManual = TRUE THEN
		p_eAct ACCESS p_UIStopper1Act2;
	ELSE
		p_eAct ACCESS ADR(eAct);
	END_IF

END_ACTION
```

#### Init.st
```iecst
(** 2019-03-25 **)
PROGRAM _INIT

	(* Always Change If Project Change *)

	//Pass Address To Global Address For External Use
	//Action, State & Status
	p_PneuNoSenTopEntStpr2Stat			:= ADR(eStat);
	p_PneuNoSenTopEntStpr2Status			:= ADR(eStatus);
	p_PneuNoSenTopEntStpr2StatTxt		:= ADR(sStatTxt);

	//Alarm
	p_PneuNoSenTopEntStpr2AlmData		:= ADR(tyAlmData);

	//Output
	p_PneuNoSenTopEntStpr2ExtCtrl		:= ADR(bExtCtrl);
	p_PneuNoSenTopEntStpr2RetCtrl		:= ADR(bRetCtrl);
	p_PneuNoSenTopEntStpr2TwoCtrlOut		:= ADR(bTwoCtrlOut);
	p_PneuNoSenTopEntStpr2Extended		:= ADR(bExtended);
	p_PneuNoSenTopEntStpr2Retracted		:= ADR(bRetracted);

	(* Always Change If Project Change *)

END_PROGRAM
```

### PneuNoSenTopMidStpr2.var - Change By Project
```iecst
(*2019-03-25*)
(**)
(*Action & State & Status*)
VAR
	p_PneuNoSenTopMidStpr2Stat : UDINT;
	p_PneuNoSenTopMidStpr2Status : UDINT;
	p_PneuNoSenTopMidStpr2StatTxt : UDINT;
END_VAR
(**)
(*Alarm*)
VAR
	p_PneuNoSenTopMidStpr2AlmData : UDINT;
END_VAR
(**)
(*Output*)
VAR
	p_PneuNoSenTopMidStpr2ExtCtrl : UDINT;
	p_PneuNoSenTopMidStpr2RetCtrl : UDINT;
	p_PneuNoSenTopMidStpr2TwoCtrlOut : UDINT;
	p_PneuNoSenTopMidStpr2Extended : UDINT;
	p_PneuNoSenTopMidStpr2Retracted : UDINT;
END_VAR
```

### Program Logical/Pneu/MagConv_Stopper/PneuNoSenTopMidStpr2 (IEC) - 1.00.0 - NtPneu v5.00.0

#### Act_Alarm.st
```iecst
(** 2019-03-25 **)
ACTION Act_Alarm:

	//Error
	IF EDGEPOS(eStatus = Error) THEN

		tyAlmData.sProgNm		:= p_sProgNm;
		tyAlmData.udiCode		:= udiStatus;
		tyAlmData.eSeverity		:= AlmSeverityError;
		tyAlmData.udiRunTime	:= tyAlmData.udiRunTime + 1;
		tyAlmData.bAlm			:= TRUE;
		tyAlmData.udiModuleNum  := udiModuleNum;
		g_sPneuNoSenProgNm		:= p_sProgNm;

		//Get Error Message
		IF tyAlmData.udiCode < 10000 OR tyAlmData.udiCode > 10099 THEN
			tyAlmData.sAlmMsg	:= 'Unknown';
			tyAlmData.sRcyMsg	:= 'Unknown';
		ELSE
			tyAlmData.sAlmMsg	:= a_tyAlmText[tyAlmData.udiCode].sAlmText;
			tyAlmData.sRcyMsg	:= a_tyAlmText[tyAlmData.udiCode].sRcyText;
		END_IF

		sStatTxt	:= tyAlmData.sAlmMsg;

	ELSIF bRstErr AND (tyAlmData.udiCode <> 0) THEN

		tyAlmData.udiCode	:= 0;
		tyAlmData.eSeverity	:= AlmSeverityNA;
		tyAlmData.sAlmMsg	:= '';
		tyAlmData.sRcyMsg	:= '';
		tyAlmData.bAlm			:= FALSE;
		sStatTxt	:= a_sStatText[eStat];

	END_IF

END_ACTION
```

#### Act_InitGlobal.st
```iecst
(** 2019-04-09 **)
ACTION Act_InitGlobal:

	(* Always Change If Project Change *)

	//Pass Data To Link
	p_bLinkOpsRun ACCESS p_OpsRun;

	p_bLinkDISafetyRlySig ACCESS p_DISafetyRlySig;

	//Pass Data To Internal Use
	p_udiRstErr ACCESS p_RstErrReset;
	p_bPrep ACCESS p_NtParamProjTopMidStprPrep2;
//	p_bDis ACCESS p_McParamTopMidStprDis;
	p_bManual ACCESS p_UIMnlMod;
	p_bTwoCtrlIn ACCESS p_NtParamTopMidStprTwoCtrlIn2;
	p_sProgNm ACCESS p_NtParamTopMidStprProgNm2;
	p_tExtDlyTm ACCESS p_NtParamTopMidStprExtDlyTm2;
	p_tRetDlyTm ACCESS p_NtParamTopMidStprRetDlyTm2;
	p_bNtSettingsLoadDone ACCESS p_StartupNtSettingsLoadDone;
	p_bPrep ACCESS p_NtParamProjMagConvLane2Prep;
	(* Always Change If Project Change *)

END_ACTION
```

#### Act_LinkAction.st
```iecst
(** 2019-04-09 **)
ACTION Act_LinkAction:

	IF p_bLinkOpsRun = TRUE AND p_OpsMagConv2StprTopMidAct <> 0  THEN
		p_eAct ACCESS p_OpsMagConv2StprTopMidAct;
	ELSIF p_bManual = TRUE THEN
		p_eAct ACCESS p_UIStopper2Act2;
	ELSE
		p_eAct ACCESS ADR(eAct);
	END_IF

END_ACTION
```

#### Init.st
```iecst
(** 2019-03-25 **)
PROGRAM _INIT

	(* Always Change If Project Change *)

	//Pass Address To Global Address For External Use
	//Action, State & Status
	p_PneuNoSenTopMidStpr2Stat			:= ADR(eStat);
	p_PneuNoSenTopMidStpr2Status			:= ADR(eStatus);
	p_PneuNoSenTopMidStpr2StatTxt		:= ADR(sStatTxt);

	//Alarm
	p_PneuNoSenTopMidStpr2AlmData		:= ADR(tyAlmData);

	//Output
	p_PneuNoSenTopMidStpr2ExtCtrl		:= ADR(bExtCtrl);
	p_PneuNoSenTopMidStpr2RetCtrl		:= ADR(bRetCtrl);
	p_PneuNoSenTopMidStpr2TwoCtrlOut		:= ADR(bTwoCtrlOut);
	p_PneuNoSenTopMidStpr2Extended		:= ADR(bExtended);
	p_PneuNoSenTopMidStpr2Retracted		:= ADR(bRetracted);

	(* Always Change If Project Change *)

END_PROGRAM
```

### PneuNoSenTopExtStpr2.var - Change By Project
```iecst
(*2019-03-25*)
(**)
(*Action & State & Status*)
VAR
	p_PneuNoSenTopExtStpr2Stat : UDINT;
	p_PneuNoSenTopExtStpr2Status : UDINT;
	p_PneuNoSenTopExtStpr2StatTxt : UDINT;
END_VAR
(**)
(*Alarm*)
VAR
	p_PneuNoSenTopExtStpr2AlmData : UDINT;
END_VAR
(**)
(*Output*)
VAR
	p_PneuNoSenTopExtStpr2ExtCtrl : UDINT;
	p_PneuNoSenTopExtStpr2RetCtrl : UDINT;
	p_PneuNoSenTopExtStpr2TwoCtrlOut : UDINT;
	p_PneuNoSenTopExtStpr2Extended : UDINT;
	p_PneuNoSenTopExtStpr2Retracted : UDINT;
END_VAR
```

### Program Logical/Pneu/MagConv_Stopper/PneuNoSenTopExtStpr2 (IEC) - 1.00.0 - NtPneu v5.00.0

#### Act_InitGlobal.st
```iecst
(** 2019-04-09 **)
ACTION Act_InitGlobal:

	(* Always Change If Project Change *)

	//Pass Data To Link
	p_bLinkOpsRun ACCESS p_OpsRun;

	p_bLinkDISafetyRlySig ACCESS p_DISafetyRlySig;

	//Pass Data To Internal Use
	p_udiRstErr ACCESS p_RstErrReset;
	p_bPrep ACCESS p_NtParamProjTopExtStprPrep2;
//	p_bDis ACCESS p_McParamTopExtStprDis;
	p_bManual ACCESS p_UIMnlMod;
	p_bTwoCtrlIn ACCESS p_NtParamTopExtStprTwoCtrlIn2;
	p_sProgNm ACCESS p_NtParamTopExtStprProgNm2;
	p_tExtDlyTm ACCESS p_NtParamTopExtStprExtDlyTm2;
	p_tRetDlyTm ACCESS p_NtParamTopExtStprRetDlyTm2;
	p_bNtSettingsLoadDone ACCESS p_StartupNtSettingsLoadDone;
	p_bPrep ACCESS p_NtParamProjMagConvLane2Prep;
	(* Always Change If Project Change *)

END_ACTION
```

#### Act_LinkAction.st
```iecst
(** 2019-04-09 **)
ACTION Act_LinkAction:

	IF p_bLinkOpsRun = TRUE AND p_OpsMagConv2StprTopExitAct <> 0  THEN
		p_eAct ACCESS p_OpsMagConv2StprTopExitAct;
	ELSIF p_bManual = TRUE THEN
		p_eAct ACCESS p_UIStopper3Act2;
	ELSE
		p_eAct ACCESS ADR(eAct);
	END_IF

END_ACTION
```

#### Init.st
```iecst
(** 2019-03-25 **)
PROGRAM _INIT

	(* Always Change If Project Change *)

	//Pass Address To Global Address For External Use
	//Action, State & Status
	p_PneuNoSenTopExtStpr2Stat			:= ADR(eStat);
	p_PneuNoSenTopExtStpr2Status			:= ADR(eStatus);
	p_PneuNoSenTopExtStpr2StatTxt		:= ADR(sStatTxt);

	//Alarm
	p_PneuNoSenTopExtStpr2AlmData		:= ADR(tyAlmData);

	//Output
	p_PneuNoSenTopExtStpr2ExtCtrl		:= ADR(bExtCtrl);
	p_PneuNoSenTopExtStpr2RetCtrl		:= ADR(bRetCtrl);
	p_PneuNoSenTopExtStpr2TwoCtrlOut		:= ADR(bTwoCtrlOut);
	p_PneuNoSenTopExtStpr2Extended		:= ADR(bExtended);
	p_PneuNoSenTopExtStpr2Retracted		:= ADR(bRetracted);

	(* Always Change If Project Change *)

END_PROGRAM
```

### PneuNoSenBtmMidStpr2.var - Change By Project
```iecst
(*2019-03-25*)
(**)
(*Action & State & Status*)
VAR
	p_PneuNoSenBtmMidStpr2Stat : UDINT;
	p_PneuNoSenBtmMidStpr2Status : UDINT;
	p_PneuNoSenBtmMidStpr2StatTxt : UDINT;
END_VAR
(**)
(*Alarm*)
VAR
	p_PneuNoSenBtmMidStpr2AlmData : UDINT;
END_VAR
(**)
(*Output*)
VAR
	p_PneuNoSenBtmMidStpr2ExtCtrl : UDINT;
	p_PneuNoSenBtmMidStpr2RetCtrl : UDINT;
	p_PneuNoSenBtmMidStpr2TwoCtrlOut : UDINT;
	p_PneuNoSenBtmMidStpr2Extended : UDINT;
	p_PneuNoSenBtmMidStpr2Retracted : UDINT;
END_VAR
```

### Program Logical/Pneu/MagConv_Stopper/PneuNoSenBtmMidStpr2 (IEC) - 1.00.0 - NtPneu v5.00.0

#### Act_Alarm.st
```iecst
(** 2019-03-25 **)
ACTION Act_Alarm:

	//Error
	IF EDGEPOS(eStatus = Error) THEN

		tyAlmData.sProgNm		:= p_sProgNm;
		tyAlmData.udiCode		:= udiStatus;
		tyAlmData.eSeverity		:= AlmSeverityError;
		tyAlmData.udiRunTime	:= tyAlmData.udiRunTime + 1;
		tyAlmData.bAlm			:= TRUE;
		tyAlmData.udiModuleNum  := udiModuleNum;
		g_sPneuNoSenProgNm		:= p_sProgNm;

		//Get Error Message
		IF tyAlmData.udiCode < 10000 OR tyAlmData.udiCode > 10099 THEN
			tyAlmData.sAlmMsg	:= 'Unknown';
			tyAlmData.sRcyMsg	:= 'Unknown';
		ELSE
			tyAlmData.sAlmMsg	:= a_tyAlmText[tyAlmData.udiCode].sAlmText;
			tyAlmData.sRcyMsg	:= a_tyAlmText[tyAlmData.udiCode].sRcyText;
		END_IF

		sStatTxt	:= tyAlmData.sAlmMsg;

	ELSIF bRstErr AND (tyAlmData.udiCode <> 0) THEN

		tyAlmData.udiCode	:= 0;
		tyAlmData.eSeverity	:= AlmSeverityNA;
		tyAlmData.sAlmMsg	:= '';
		tyAlmData.sRcyMsg	:= '';
		tyAlmData.bAlm			:= FALSE;
		sStatTxt	:= a_sStatText[eStat];

	END_IF

END_ACTION
```

#### Act_InitGlobal.st
```iecst
(** 2019-04-09 **)
ACTION Act_InitGlobal:

	(* Always Change If Project Change *)

	//Pass Data To Link
	p_bLinkOpsRun ACCESS p_OpsRun;

	p_bLinkDISafetyRlySig ACCESS p_DISafetyRlySig;

	//Pass Data To Internal Use
	p_udiRstErr ACCESS p_RstErrReset;
	p_bPrep ACCESS p_NtParamProjBtmMidStprPrep2;
//	p_bDis ACCESS p_McParamBtmMidStprDis;
	p_bManual ACCESS p_UIMnlMod;
	p_bTwoCtrlIn ACCESS p_NtParamBtmMidStprTwoCtrlIn2;
	p_sProgNm ACCESS p_NtParamBtmMidStprProgNm2;
	p_tExtDlyTm ACCESS p_NtParamBtmMidStprExtDlyTm2;
	p_tRetDlyTm ACCESS p_NtParamBtmMidStprRetDlyTm2;
	p_bNtSettingsLoadDone ACCESS p_StartupNtSettingsLoadDone;
	p_bPrep ACCESS p_NtParamProjMagConvLane2Prep;
	(* Always Change If Project Change *)

END_ACTION
```

#### Act_LinkAction.st
```iecst
(** 2019-04-09 **)
ACTION Act_LinkAction:

	IF p_bLinkOpsRun = TRUE AND p_OpsMagConv2StprBtmMidAct <> 0 THEN
		p_eAct ACCESS p_OpsMagConv2StprBtmMidAct;
	ELSIF p_bManual = TRUE THEN
		p_eAct ACCESS p_UIStopper4Act2;
	ELSE
		p_eAct ACCESS ADR(eAct);
	END_IF

END_ACTION
```

#### Init.st
```iecst
(** 2019-03-25 **)
PROGRAM _INIT

	(* Always Change If Project Change *)

	//Pass Address To Global Address For External Use
	//Action, State & Status
	p_PneuNoSenBtmMidStpr2Stat			:= ADR(eStat);
	p_PneuNoSenBtmMidStpr2Status			:= ADR(eStatus);
	p_PneuNoSenBtmMidStpr2StatTxt		:= ADR(sStatTxt);

	//Alarm
	p_PneuNoSenBtmMidStpr2AlmData		:= ADR(tyAlmData);

	//Output
	p_PneuNoSenBtmMidStpr2ExtCtrl		:= ADR(bExtCtrl);
	p_PneuNoSenBtmMidStpr2RetCtrl		:= ADR(bRetCtrl);
	p_PneuNoSenBtmMidStpr2TwoCtrlOut		:= ADR(bTwoCtrlOut);
	p_PneuNoSenBtmMidStpr2Extended		:= ADR(bExtended);
	p_PneuNoSenBtmMidStpr2Retracted		:= ADR(bRetracted);

	(* Always Change If Project Change *)

END_PROGRAM
```

### PneuNoSenBtmExtStpr2.var - Change By Project
```iecst
(*2019-03-25*)
(**)
(*Action & State & Status*)
VAR
	p_PneuNoSenBtmExtStpr2Stat : UDINT;
	p_PneuNoSenBtmExtStpr2Status : UDINT;
	p_PneuNoSenBtmExtStpr2StatTxt : UDINT;
END_VAR
(**)
(*Alarm*)
VAR
	p_PneuNoSenBtmExtStpr2AlmData : UDINT;
END_VAR
(**)
(*Output*)
VAR
	p_PneuNoSenBtmExtStpr2ExtCtrl : UDINT;
	p_PneuNoSenBtmExtStpr2RetCtrl : UDINT;
	p_PneuNoSenBtmExtStpr2TwoCtrlOut : UDINT;
	p_PneuNoSenBtmExtStpr2Extended : UDINT;
	p_PneuNoSenBtmExtStpr2Retracted : UDINT;
END_VAR
```

### Program Logical/Pneu/MagConv_Stopper/PneuNoSenBtmExtStpr2 (IEC) - 1.00.0 - NtPneu v5.00.0

#### Act_InitGlobal.st
```iecst
(** 2019-04-09 **)
ACTION Act_InitGlobal:

	(* Always Change If Project Change *)

	//Pass Data To Link
	p_bLinkOpsRun ACCESS p_OpsRun;

	p_bLinkDISafetyRlySig ACCESS p_DISafetyRlySig;

	//Pass Data To Internal Use
	p_udiRstErr ACCESS p_RstErrReset;
	p_bPrep ACCESS p_NtParamProjBtmExtStprPrep2;
//	p_bDis ACCESS p_McParamBtmExtStprDis;
	p_bManual ACCESS p_UIMnlMod;
	p_bTwoCtrlIn ACCESS p_NtParamBtmExtStprTwoCtrlIn2;
	p_sProgNm ACCESS p_NtParamBtmExtStprProgNm2;
	p_tExtDlyTm ACCESS p_NtParamBtmExtStprExtDlyTm2;
	p_tRetDlyTm ACCESS p_NtParamBtmExtStprRetDlyTm2;
	p_bNtSettingsLoadDone ACCESS p_StartupNtSettingsLoadDone;
	p_bPrep ACCESS p_NtParamProjMagConvLane2Prep;
	(* Always Change If Project Change *)

END_ACTION
```

#### Act_LinkAction.st
```iecst
(** 2019-04-09 **)
ACTION Act_LinkAction:

	IF p_bLinkOpsRun = TRUE AND p_OpsMagConv2StprBtmExitAct <> 0 THEN
		p_eAct ACCESS p_OpsMagConv2StprBtmExitAct;
	ELSIF p_bManual = TRUE THEN
		p_eAct ACCESS p_UIStopper5Act2;
	ELSE
		p_eAct ACCESS ADR(eAct);
	END_IF

END_ACTION
```

#### Init.st
```iecst
(** 2019-03-25 **)
PROGRAM _INIT

	(* Always Change If Project Change *)

	//Pass Address To Global Address For External Use
	//Action, State & Status
	p_PneuNoSenBtmExtStpr2Stat			:= ADR(eStat);
	p_PneuNoSenBtmExtStpr2Status			:= ADR(eStatus);
	p_PneuNoSenBtmExtStpr2StatTxt		:= ADR(sStatTxt);

	//Alarm
	p_PneuNoSenBtmExtStpr2AlmData		:= ADR(tyAlmData);

	//Output
	p_PneuNoSenBtmExtStpr2ExtCtrl		:= ADR(bExtCtrl);
	p_PneuNoSenBtmExtStpr2RetCtrl		:= ADR(bRetCtrl);
	p_PneuNoSenBtmExtStpr2TwoCtrlOut		:= ADR(bTwoCtrlOut);
	p_PneuNoSenBtmExtStpr2Extended		:= ADR(bExtended);
	p_PneuNoSenBtmExtStpr2Retracted		:= ADR(bRetracted);

	(* Always Change If Project Change *)

END_PROGRAM
```

### Program Logical/Pneu/Pneu2SenInShutter

#### InputRef.var
```iecst
(*2019-03-25*)
(**)
(*General*)
VAR
	p_eAct : REFERENCE TO ePneuAction;
	p_udiRstErr : REFERENCE TO UDINT;
	p_bPrep : REFERENCE TO BOOL;
	p_bEn : REFERENCE TO BOOL;
	p_bDis : REFERENCE TO BOOL;
END_VAR
(**)
(*Configuration*)
VAR
	p_bUISimu : REFERENCE TO BOOL;
	p_bManual : REFERENCE TO BOOL;
	p_bSimu : REFERENCE TO BOOL;
	p_bTwoCtrlIn : REFERENCE TO BOOL;
	p_bExtSafetySen : REFERENCE TO BOOL;
	p_bRetSafetySen : REFERENCE TO BOOL;
	p_sProgNm : REFERENCE TO STRING[15];
	p_tExtTO : REFERENCE TO TIME;
	p_tRetTO : REFERENCE TO TIME;
	p_bNtSettingsLoadDone : REFERENCE TO BOOL;
END_VAR
(**)
(*Input*)
VAR
	p_bExtSen : REFERENCE TO BOOL;
	p_bRetSen : REFERENCE TO BOOL;
END_VAR
```

#### InputRef_Link.var
```iecst
(*2019-04-09*)
(**)
(*External*)
VAR
	p_bLinkOpsRun : REFERENCE TO BOOL;
END_VAR
(**)
VAR
	p_bLinkDISafetyRlySig : REFERENCE TO BOOL;
	p_bLinkInitOpsTravULDone : REFERENCE TO BOOL;
	p_bLinkMcParamInShutDis : REFERENCE TO BOOL;
END_VAR
```

#### Act_InitGlobal.st
```iecst
(** 2019-04-09 **)
ACTION Act_InitGlobal:

	(* Always Change If Project Change *)

	//Pass Data To Link
	p_bLinkOpsRun ACCESS p_OpsRun;

	p_bLinkDISafetyRlySig ACCESS p_DISafetyRlySig;
	p_bLinkInitOpsTravULDone ACCESS p_OpsTravLifULInitDone;
	p_bLinkMcParamInShutDis ACCESS p_McParamInShutterDis;

	//Pass Data To Internal Use
	p_udiRstErr ACCESS p_RstErrReset;
	p_bPrep ACCESS p_NtParamProjInletShutPrep;
	//	p_bDis ACCESS p_McParamInShutterDis;
	p_bUISimu ACCESS p_UISimuMod;
	p_bManual ACCESS p_UIMnlMod;
	p_bSimu ACCESS p_UISimuMod;
	p_bTwoCtrlIn ACCESS p_NtParamInShutterTwoCtrlIn;
	p_sProgNm ACCESS p_NtParamInShutterProgNm;
	p_bExtSen ACCESS p_DIInShutterCloseRS;
	p_bRetSen ACCESS p_DIInShutterOpenRS;
	p_tExtTO ACCESS p_NtParamInShutterExtTO;
	p_tRetTO ACCESS p_NtParamInShutterRetTO;
	p_bNtSettingsLoadDone ACCESS p_StartupNtSettingsLoadDone;

	(* Always Change If Project Change *)

END_ACTION
```

#### Act_LinkAction.st
```iecst
(** 2019-04-09 **)
ACTION Act_LinkAction:

	IF p_bLinkOpsRun = TRUE THEN
		p_eAct ACCESS p_OpsTravLifULInletPneuAct;
	ELSIF p_bManual = TRUE OR p_bUISimu THEN
		p_eAct ACCESS p_UIInShutterAct;
	ELSE
		p_eAct ACCESS ADR(eAct);
	END_IF

END_ACTION
```

#### Act_LinkEn.st
```iecst
(** 2019-01-11 **)
ACTION Act_LinkEn:

	//Link bPrep, bEn & bDis
	IF p_bLinkOpsRun THEN
		p_bDis := p_bLinkMcParamInShutDis AND p_bLinkInitOpsTravULDone;
	ELSE
		p_bDis := FALSE;
	END_IF

END_ACTION
```

### Program Logical/Pneu/Pneu2SenMag1AWEngage

#### Act_InitGlobal.st
```iecst
(** 2019-04-09 **)
ACTION Act_InitGlobal:

	(* Always Change If Project Change *)

	//Pass Data To Link
	p_bLinkOpsRun ACCESS p_OpsRun;

	p_bLinkDISafetyRlySig ACCESS p_DISafetyRlySig;

	//Pass Data To Internal Use
	p_udiRstErr ACCESS p_RstErrReset;
	p_bPrep ACCESS p_NtParamProjMagAWPrep;
	p_bDis ACCESS p_McParamMagAWDis;
	p_bManual ACCESS p_UIMnlMod;
	p_bTwoCtrlIn ACCESS p_NtParamMag1AWEngageTwoCtrlIn;
	p_sProgNm ACCESS p_NtParamMag1AWEngageProgNm;
	p_bExtSen ACCESS p_DIMag1WallEngageRS;
	p_bRetSen ACCESS p_DIMag1WallDisengageRS;
	p_tExtTO ACCESS p_NtParamMag1AWEngageExtTO;
	p_tRetTO ACCESS p_NtParamMag1AWEngageRetTO;
	p_bNtSettingsLoadDone ACCESS p_StartupNtSettingsLoadDone;

	(* Always Change If Project Change *)

END_ACTION
```

#### Act_LinkAction.st
```iecst
(** 2019-04-09 **)
ACTION Act_LinkAction:

	IF p_bLinkOpsRun = TRUE THEN
		p_eAct ACCESS p_OpsMagConvUL1MagAWEngageAct;
	ELSIF p_bManual = TRUE THEN
		p_eAct ACCESS p_UIMag1AWEngageAct;
	ELSE
		p_eAct ACCESS ADR(eAct);
	END_IF

END_ACTION
```

#### Init.st
```iecst
(** 2019-03-25 **)
PROGRAM _INIT

	(* Always Change If Project Change *)

	//Pass Address To Global Address For External Use
	//Action, State & Status
	p_Pneu2SMag1AWEngageStat	:= ADR(eStat);
	p_Pneu2SMag1AWEngageStatus	:= ADR(eStatus);
	p_Pneu2SMag1AWEngageStatTxt	:= ADR(sStatTxt);

	//Alarm
	p_Pneu2SMag1AWEngageAlmData	:= ADR(tyAlmData);

	//Output
	p_Pneu2SMag1AWEngageExtCtrl		:= ADR(bExtCtrl);
	p_Pneu2SMag1AWEngageRetCtrl		:= ADR(bRetCtrl);
	p_Pneu2SMag1AWEngageTwoCtrlOut	:= ADR(bTwoCtrlOut);
	p_Pneu2SMag1AWEngageExtended	:= ADR(bExtended);
	p_Pneu2SMag1AWEngageRetracted	:= ADR(bRetracted);

	(* Always Change If Project Change *)

END_PROGRAM
```

### Program Logical/Pneu/Pneu2SenMag1SafetyBar

#### Act_Alarm.st
```iecst
(** 2019-03-25 **)
ACTION Act_Alarm:

	//Error
	IF EDGEPOS(eStatus = Error) THEN

		tyAlmData.sProgNm		:= p_sProgNm;
		tyAlmData.udiCode		:= udiStatus;
		tyAlmData.eSeverity		:= AlmSeverityError;
		tyAlmData.udiRunTime	:= tyAlmData.udiRunTime + 1;
		tyAlmData.bAlm			:= TRUE;
		tyAlmData.udiModuleNum  := udiModuleNum;
		g_sPneu2SenProgNm		:= p_sProgNm;

		//Get Error Message
		IF tyAlmData.udiCode < 10000 OR tyAlmData.udiCode > 10099 THEN
			tyAlmData.sAlmMsg	:= 'Unknown';
			tyAlmData.sRcyMsg	:= 'Unknown';
		ELSE
			tyAlmData.sAlmMsg	:= a_tyAlmText[tyAlmData.udiCode].sAlmText;
			tyAlmData.sRcyMsg	:= a_tyAlmText[tyAlmData.udiCode].sRcyText;
		END_IF

		sStatTxt	:= tyAlmData.sAlmMsg;

	ELSIF bRstErr AND (tyAlmData.udiCode <> 0) THEN

		tyAlmData.udiCode	:= 0;
		tyAlmData.eSeverity	:= AlmSeverityNA;
		tyAlmData.sAlmMsg	:= '';
		tyAlmData.sRcyMsg	:= '';
		tyAlmData.bAlm			:= FALSE;
		sStatTxt	:= a_sStatText[eStat];

	END_IF

END_ACTION
```

#### Act_InitGlobal.st
```iecst
(** 2019-04-09 **)
ACTION Act_InitGlobal:

	(* Always Change If Project Change *)

	//Pass Data To Link
	p_bLinkOpsRun ACCESS p_OpsRun;

	p_bLinkDISafetyRlySig ACCESS p_DISafetyRlySig;
	p_bMagRcpCurrRcpSBarDisabled ACCESS p_MagRcpCurrRcpSBarDisabled;

	//Pass Data To Internal Use
	p_udiRstErr ACCESS p_RstErrReset;
	p_bPrep ACCESS p_NtParamProjMagSafetyBarPrep;
//	p_bDis ACCESS p_McParamMagAWDis;
	p_bManual ACCESS p_UIMnlMod;
	p_bTwoCtrlIn ACCESS p_NtParamMag1SafetyBarTwoCtrlIn;
	p_sProgNm ACCESS p_NtParamMag1SafetyBarProgNm;
	p_bExtSen ACCESS p_DIMag1SafetyBarExtRS;
	p_bRetSen ACCESS p_DIMag1SafetyBarRetRS;
	p_tExtTO ACCESS p_NtParamMag1SafetyBarExtTO;
	p_tRetTO ACCESS p_NtParamMag1SafetyBarRetTO;
	p_bNtSettingsLoadDone ACCESS p_StartupNtSettingsLoadDone;

	(* Always Change If Project Change *)

END_ACTION
```

#### Act_Link.st
```iecst
(** 2019-03-29 **)
ACTION Act_Link:

	IF p_bLinkDISafetyRlySig = FALSE THEN
		bExtCtrl	:= FALSE;
		bRetCtrl	:= FALSE;
		bExtended	:= FALSE;
		bRetracted	:= FALSE;
	END_IF

END_ACTION
```

#### Act_LinkAction.st
```iecst
(** 2019-04-09 **)
ACTION Act_LinkAction:

	IF p_bLinkOpsRun = TRUE THEN
		p_eAct ACCESS p_OpsMagConvUL1SafetyBarAct;
	ELSIF p_bManual = TRUE THEN
		p_eAct ACCESS p_UIMag1SafetyBarAct;
	ELSE
		p_eAct ACCESS ADR(eAct);
	END_IF

END_ACTION
```

#### Init.st
```iecst
(** 2019-03-25 **)
PROGRAM _INIT

	(* Always Change If Project Change *)

	//Pass Address To Global Address For External Use
	//Action, State & Status
	p_Pneu2SMag1SafetyBarStat		:= ADR(eStat);
	p_Pneu2SMag1SafetyBarStatus		:= ADR(eStatus);
	p_Pneu2SMag1SafetyBarStatTxt	:= ADR(sStatTxt);

	//Alarm
	p_Pneu2SMag1SafetyBarAlmData	:= ADR(tyAlmData);

	//Output
	p_Pneu2SMag1SafetyBarExtCtrl	:= ADR(bExtCtrl);
	p_Pneu2SMag1SafetyBarRetCtrl	:= ADR(bRetCtrl);
	p_Pneu2SMag1SafetyBarTwoCtrlOut	:= ADR(bTwoCtrlOut);
	p_Pneu2SMag1SafetyBarExtended	:= ADR(bExtended);
	p_Pneu2SMag1SafetyBarRetracted	:= ADR(bRetracted);

	(* Always Change If Project Change *)

END_PROGRAM
```

### Program Logical/Pneu/Pneu2SenMag2AWEngage

#### Act_InitGlobal.st
```iecst
(** 2019-04-09 **)
ACTION Act_InitGlobal:

	(* Always Change If Project Change *)

	//Pass Data To Link
	p_bLinkOpsRun ACCESS p_OpsRun;

	p_bLinkDISafetyRlySig ACCESS p_DISafetyRlySig;

	//Pass Data To Internal Use
	p_udiRstErr ACCESS p_RstErrReset;
	p_bPrep ACCESS p_NtParamProjMagAWPrep;
	p_bDis ACCESS p_McParamMagAWDis;
	p_bManual ACCESS p_UIMnlMod;
	p_bTwoCtrlIn ACCESS p_NtParamMag2AWEngageTwoCtrlIn;
	p_sProgNm ACCESS p_NtParamMag2AWEngageProgNm;
	p_bExtSen ACCESS p_DIMag2WallEngageRS;
	p_bRetSen ACCESS p_DIMag2WallDisengageRS;
	p_tExtTO ACCESS p_NtParamMag2AWEngageExtTO;
	p_tRetTO ACCESS p_NtParamMag2AWEngageRetTO;
	p_bNtSettingsLoadDone ACCESS p_StartupNtSettingsLoadDone;

	(* Always Change If Project Change *)

END_ACTION
```

#### Act_LinkAction.st
```iecst
(** 2019-04-09 **)
ACTION Act_LinkAction:

	IF p_bLinkOpsRun = TRUE THEN
		p_eAct ACCESS p_OpsMagConvUL2MagAWEngageAct;
	ELSIF p_bManual = TRUE THEN
		p_eAct ACCESS p_UIMag2AWEngageAct;
	ELSE
		p_eAct ACCESS ADR(eAct);
	END_IF

END_ACTION
```

#### Init.st
```iecst
(** 2019-03-25 **)
PROGRAM _INIT

	(* Always Change If Project Change *)

	//Pass Address To Global Address For External Use
	//Action, State & Status
	p_Pneu2SMag2AWEngageStat	:= ADR(eStat);
	p_Pneu2SMag2AWEngageStatus	:= ADR(eStatus);
	p_Pneu2SMag2AWEngageStatTxt	:= ADR(sStatTxt);

	//Alarm
	p_Pneu2SMag2AWEngageAlmData	:= ADR(tyAlmData);

	//Output
	p_Pneu2SMag2AWEngageExtCtrl		:= ADR(bExtCtrl);
	p_Pneu2SMag2AWEngageRetCtrl		:= ADR(bRetCtrl);
	p_Pneu2SMag2AWEngageTwoCtrlOut	:= ADR(bTwoCtrlOut);
	p_Pneu2SMag2AWEngageExtended	:= ADR(bExtended);
	p_Pneu2SMag2AWEngageRetracted	:= ADR(bRetracted);

	(* Always Change If Project Change *)

END_PROGRAM
```

### Program Logical/Pneu/Pneu2SenMag2SafetyBar

#### InputRef_Link.var
```iecst
(*2019-04-09*)
(**)
(*External*)
VAR
	p_bLinkOpsRun : REFERENCE TO BOOL;
END_VAR
(**)
VAR
	p_bLinkDISafetyRlySig : REFERENCE TO BOOL;
	p_bMagRcpCurrRcpSBarDisabled : REFERENCE TO BOOL;
END_VAR
```

#### Act_InitGlobal.st
```iecst
(** 2019-04-09 **)
ACTION Act_InitGlobal:

	(* Always Change If Project Change *)

	//Pass Data To Link
	p_bLinkOpsRun ACCESS p_OpsRun;

	p_bLinkDISafetyRlySig ACCESS p_DISafetyRlySig;
	p_bMagRcpCurrRcpSBarDisabled ACCESS p_MagRcpCurrRcpSBarDisabled;

	//Pass Data To Internal Use
	p_udiRstErr ACCESS p_RstErrReset;
	p_bPrep ACCESS p_NtParamProjMagSafetyBarPrep;
//	p_bDis ACCESS p_McParamMagAWDis;
	p_bManual ACCESS p_UIMnlMod;
	p_bTwoCtrlIn ACCESS p_NtParamMag2SafetyBarTwoCtrlIn;
	p_sProgNm ACCESS p_NtParamMag2SafetyBarProgNm;
	p_bExtSen ACCESS p_DIMag2SafetyBarExtRS;
	p_bRetSen ACCESS p_DIMag2SafetyBarRetRS;
	p_tExtTO ACCESS p_NtParamMag2SafetyBarExtTO;
	p_tRetTO ACCESS p_NtParamMag2SafetyBarRetTO;
	p_bNtSettingsLoadDone ACCESS p_StartupNtSettingsLoadDone;

	(* Always Change If Project Change *)

END_ACTION
```

#### Act_LinkAction.st
```iecst
(** 2019-04-09 **)
ACTION Act_LinkAction:

	IF p_bLinkOpsRun = TRUE THEN
		p_eAct ACCESS p_OpsMagConvUL2SafetyBarAct;
	ELSIF p_bManual = TRUE THEN
		p_eAct ACCESS p_UIMag2SafetyBarAct;
	ELSE
		p_eAct ACCESS ADR(eAct);
	END_IF

END_ACTION
```

#### Act_LinkEn.st
```iecst
(** 2019-01-11 **)
ACTION Act_LinkEn:

	//Link bPrep, bEn & bDis
	IF p_bLinkOpsRun AND p_bPrep THEN
		p_bDis := p_bMagRcpCurrRcpSBarDisabled;
	ELSE
		p_bDis := FALSE;
	END_IF

END_ACTION
```

#### Init.st
```iecst
(** 2019-03-25 **)
PROGRAM _INIT

	(* Always Change If Project Change *)

	//Pass Address To Global Address For External Use
	//Action, State & Status
	p_Pneu2SMag2SafetyBarStat		:= ADR(eStat);
	p_Pneu2SMag2SafetyBarStatus		:= ADR(eStatus);
	p_Pneu2SMag2SafetyBarStatTxt	:= ADR(sStatTxt);

	//Alarm
	p_Pneu2SMag2SafetyBarAlmData	:= ADR(tyAlmData);

	//Output
	p_Pneu2SMag2SafetyBarExtCtrl	:= ADR(bExtCtrl);
	p_Pneu2SMag2SafetyBarRetCtrl	:= ADR(bRetCtrl);
	p_Pneu2SMag2SafetyBarTwoCtrlOut	:= ADR(bTwoCtrlOut);
	p_Pneu2SMag2SafetyBarExtended	:= ADR(bExtended);
	p_Pneu2SMag2SafetyBarRetracted	:= ADR(bRetracted);

	(* Always Change If Project Change *)

END_PROGRAM
```

### Program Logical/Pneu/Pneu2SenMag3AWEngage

#### InputRef_Link.var
```iecst
(*2019-04-09*)
(**)
(*External*)
VAR
	p_bLinkOpsRun : REFERENCE TO BOOL;
END_VAR
(**)
VAR
	p_bLinkNtParamProjMagAWPrep : REFERENCE TO BOOL;
	p_bLinkNtParamProjMag : REFERENCE TO eULMag;
END_VAR
(**)
VAR
	p_bLinkDISafetyRlySig : REFERENCE TO BOOL;
END_VAR
```

#### Act_InitGlobal.st
```iecst
(** 2019-04-09 **)
ACTION Act_InitGlobal:

	(* Always Change If Project Change *)

	//Pass Data To Link
	p_bLinkOpsRun ACCESS p_OpsRun;

	p_bLinkNtParamProjMagAWPrep ACCESS p_NtParamProjMagAWPrep;
	p_bLinkNtParamProjMag ACCESS p_NtParamProjMag;

	p_bLinkDISafetyRlySig ACCESS p_DISafetyRlySig;

	//Pass Data To Internal Use
	p_udiRstErr ACCESS p_RstErrReset;
	p_bDis ACCESS p_McParamMagAWDis;
	p_bManual ACCESS p_UIMnlMod;
	p_bTwoCtrlIn ACCESS p_NtParamMag3AWEngageTwoCtrlIn;
	p_sProgNm ACCESS p_NtParamMag3AWEngageProgNm;
	p_bExtSen ACCESS p_DIMag3WallEngageRS;
	p_bRetSen ACCESS p_DIMag3WallDisengageRS;
	p_tExtTO ACCESS p_NtParamMag3AWEngageExtTO;
	p_tRetTO ACCESS p_NtParamMag3AWEngageRetTO;
	p_bNtSettingsLoadDone ACCESS p_StartupNtSettingsLoadDone;

	(* Always Change If Project Change *)

END_ACTION
```

#### Act_LinkAction.st
```iecst
(** 2019-04-09 **)
ACTION Act_LinkAction:

	IF p_bLinkOpsRun = TRUE THEN
		p_eAct ACCESS p_OpsMagConvUL3MagAWEngageAct;
	ELSIF p_bManual = TRUE THEN
		p_eAct ACCESS p_UIMag3AWEngageAct;
	ELSE
		p_eAct ACCESS ADR(eAct);
	END_IF

END_ACTION
```

#### Act_LinkEn.st
```iecst
(** 2019-01-11 **)
ACTION Act_LinkEn:

	//Link bPrep, bEn & bDis
	p_bPrep	:= p_bLinkNtParamProjMagAWPrep AND p_bLinkNtParamProjMag = ULMagTriple;

END_ACTION
```

#### Init.st
```iecst
(** 2019-03-25 **)
PROGRAM _INIT

	(* Always Change If Project Change *)

	//Pass Address To Global Address For External Use
	//Action, State & Status
	p_Pneu2SMag3AWEngageStat	:= ADR(eStat);
	p_Pneu2SMag3AWEngageStatus	:= ADR(eStatus);
	p_Pneu2SMag3AWEngageStatTxt	:= ADR(sStatTxt);

	//Alarm
	p_Pneu2SMag3AWEngageAlmData	:= ADR(tyAlmData);

	//Output
	p_Pneu2SMag3AWEngageExtCtrl		:= ADR(bExtCtrl);
	p_Pneu2SMag3AWEngageRetCtrl		:= ADR(bRetCtrl);
	p_Pneu2SMag3AWEngageTwoCtrlOut	:= ADR(bTwoCtrlOut);
	p_Pneu2SMag3AWEngageExtended	:= ADR(bExtended);
	p_Pneu2SMag3AWEngageRetracted	:= ADR(bRetracted);

	(* Always Change If Project Change *)

END_PROGRAM
```

### Program Logical/Pneu/Pneu2SenMag3SafetyBar

#### InputRef_Link.var
```iecst
(*2019-04-09*)
(**)
(*External*)
VAR
	p_bLinkOpsRun : REFERENCE TO BOOL;
END_VAR
(**)
VAR
	p_bLinkNtPrmProjMagSafetyBarPrep : REFERENCE TO BOOL;
	p_bLinkNtPrmProjMag : REFERENCE TO eULMag;
END_VAR
(**)
VAR
	p_bLinkDISafetyRlySig : REFERENCE TO BOOL;
	p_bMagRcpCurrRcpSBarDisabled : REFERENCE TO BOOL;
END_VAR
```

#### Act_InitGlobal.st
```iecst
(** 2019-04-09 **)
ACTION Act_InitGlobal:

	(* Always Change If Project Change *)

	//Pass Data To Link
	p_bLinkOpsRun ACCESS p_OpsRun;

	p_bLinkNtPrmProjMagSafetyBarPrep ACCESS p_NtParamProjMagSafetyBarPrep;
	p_bLinkNtPrmProjMag ACCESS p_NtParamProjMag;

	p_bLinkDISafetyRlySig ACCESS p_DISafetyRlySig;
	p_bMagRcpCurrRcpSBarDisabled ACCESS p_MagRcpCurrRcpSBarDisabled;

	//Pass Data To Internal Use
	p_udiRstErr ACCESS p_RstErrReset;
//	p_bDis ACCESS p_McParamMagAWDis;
	p_bManual ACCESS p_UIMnlMod;
	p_bTwoCtrlIn ACCESS p_NtParamMag3SafetyBarTwoCtrlIn;
	p_sProgNm ACCESS p_NtParamMag3SafetyBarProgNm;
	p_bExtSen ACCESS p_DIMag3SafetyBarExtRS;
	p_bRetSen ACCESS p_DIMag3SafetyBarRetRS;
	p_tExtTO ACCESS p_NtParamMag3SafetyBarExtTO;
	p_tRetTO ACCESS p_NtParamMag3SafetyBarRetTO;
	p_bNtSettingsLoadDone ACCESS p_StartupNtSettingsLoadDone;

	(* Always Change If Project Change *)

END_ACTION
```

#### Act_LinkAction.st
```iecst
(** 2019-04-09 **)
ACTION Act_LinkAction:

	IF p_bLinkOpsRun = TRUE THEN
		p_eAct ACCESS p_OpsMagConvUL3SafetyBarAct;
	ELSIF p_bManual = TRUE THEN
		p_eAct ACCESS p_UIMag3SafetyBarAct;
	ELSE
		p_eAct ACCESS ADR(eAct);
	END_IF

END_ACTION
```

#### Act_LinkEn.st
```iecst
(** 2019-01-11 **)
ACTION Act_LinkEn:

	//Link bPrep, bEn & bDis
	p_bPrep	:= p_bLinkNtPrmProjMagSafetyBarPrep AND p_bLinkNtPrmProjMag = ULMagTriple;

	IF p_bLinkOpsRun AND p_bPrep THEN
		p_bDis := p_bMagRcpCurrRcpSBarDisabled;
	ELSE
		p_bDis := FALSE;
	END_IF

END_ACTION
```

#### Init.st
```iecst
(** 2019-03-25 **)
PROGRAM _INIT

	(* Always Change If Project Change *)

	//Pass Address To Global Address For External Use
	//Action, State & Status
	p_Pneu2SMag3SafetyBarStat		:= ADR(eStat);
	p_Pneu2SMag3SafetyBarStatus		:= ADR(eStatus);
	p_Pneu2SMag3SafetyBarStatTxt	:= ADR(sStatTxt);

	//Alarm
	p_Pneu2SMag3SafetyBarAlmData	:= ADR(tyAlmData);

	//Output
	p_Pneu2SMag3SafetyBarExtCtrl	:= ADR(bExtCtrl);
	p_Pneu2SMag3SafetyBarRetCtrl	:= ADR(bRetCtrl);
	p_Pneu2SMag3SafetyBarTwoCtrlOut	:= ADR(bTwoCtrlOut);
	p_Pneu2SMag3SafetyBarExtended	:= ADR(bExtended);
	p_Pneu2SMag3SafetyBarRetracted	:= ADR(bRetracted);

	(* Always Change If Project Change *)

END_PROGRAM
```

### Program Logical/Pneu/Pneu2SenOutShutter

#### InputRef.var
```iecst
(*2019-03-25*)
(**)
(*General*)
VAR
	p_eAct : REFERENCE TO ePneuAction;
	p_udiRstErr : REFERENCE TO UDINT;
	p_bPrep : REFERENCE TO BOOL;
	p_bEn : REFERENCE TO BOOL;
	p_bDis : REFERENCE TO BOOL;
END_VAR
(**)
(*Configuration*)
VAR
	p_bUISimu : REFERENCE TO BOOL;
	p_bManual : REFERENCE TO BOOL;
	p_bSimu : REFERENCE TO BOOL;
	p_bTwoCtrlIn : REFERENCE TO BOOL;
	p_bExtSafetySen : REFERENCE TO BOOL;
	p_bRetSafetySen : REFERENCE TO BOOL;
	p_sProgNm : REFERENCE TO STRING[15];
	p_tExtTO : REFERENCE TO TIME;
	p_tRetTO : REFERENCE TO TIME;
	p_bNtSettingsLoadDone : REFERENCE TO BOOL;
	p_bNtParamProjLifter2Prep : REFERENCE TO BOOL;
END_VAR
(**)
(*Input*)
VAR
	p_bExtSen : REFERENCE TO BOOL;
	p_bRetSen : REFERENCE TO BOOL;
END_VAR
```

#### Act_InitGlobal.st
```iecst
(** 2019-04-09 **)
ACTION Act_InitGlobal:

	(* Always Change If Project Change *)

	//Pass Data To Link
	p_bLinkOpsRun ACCESS p_OpsRun;

	p_bLinkDISafetyRlySig ACCESS p_DISafetyRlySig;
	p_bLinkDIConvClrSen ACCESS p_DIConvClrSen;
	p_bConvPusherReachedRetSlw ACCESS p_PshrConvPshrRetAllwTrav;
	p_bLinkDIPusherRetRS ACCESS p_DIPusherRetRS;
	p_eLinkLifterBtmStat ACCESS p_LifterBtmStat;
	p_eLinkLifterBtmStatus ACCESS p_LifterBtmStatus;
	p_eLinkLifter2Stat ACCESS p_Lifter2Stat;
	p_eLinkLifter2Status ACCESS p_Lifter2Status;

	//Pass Data To Internal Use
	p_udiRstErr ACCESS p_RstErrReset;
	p_bPrep ACCESS p_NtParamProjOutletShutPrep;
	p_bUISimu ACCESS p_UISimuMod;
	p_bManual ACCESS p_UIMnlMod;
	p_bSimu ACCESS p_SimuRun;
	p_bTwoCtrlIn ACCESS p_NtParamOutShutterTwoCtrlIn;
	p_sProgNm ACCESS p_NtParamOutShutterProgNm;
	p_bExtSen ACCESS p_DIOutShutterCloseRS;
	p_bRetSen ACCESS p_DIOutShutterOpenRS;
	p_tExtTO ACCESS p_NtParamOutShutterExtTO;
	p_tRetTO ACCESS p_NtParamOutShutterRetTO;
	p_bNtSettingsLoadDone ACCESS p_StartupNtSettingsLoadDone;
	p_bNtParamProjLifter2Prep ACCESS p_NtParamProjLifter2Prep;
	(* Always Change If Project Change *)

END_ACTION
```

#### Act_LinkAction.st
```iecst
(** 2019-04-09 **)
ACTION Act_LinkAction:

	IF p_bLinkOpsRun = TRUE THEN
		IF p_bNtParamProjLifter2Prep = FALSE  THEN
//			IF p_eLinkLifterBtmStat = LifterActIdle AND p_eLinkLifterBtmStatus <> Busy  THEN
				p_eAct ACCESS p_OpsTravLifULOutletPneuAct;
//			ELSE
//				p_eAct ACCESS ADR(eAct);
//			END_IF
		ELSE
			IF p_eLinkLifterBtmStat = LifterActIdle AND p_eLinkLifterBtmStatus <> Busy AND p_eLinkLifter2Stat = LifterActIdle AND p_eLinkLifter2Status <> Busy  THEN // p_eLinkLifter2Status <> Busy
				p_eAct ACCESS p_OpsTravLifULOutletPneuAct;
			ELSE
				p_eAct ACCESS ADR(eAct);
			END_IF
		END_IF
	ELSIF p_bManual = TRUE OR p_bUISimu THEN
		p_eAct ACCESS p_UIOutShutterAct;
	ELSIF p_bSimu THEN
		p_eAct ACCESS p_Simu1OutShutterAct;
	ELSE
		p_eAct ACCESS ADR(eAct);
	END_IF

END_ACTION
```

### Program Logical/Pneu/Pneu2SenOutShutter2
